   1:  PR[91,3] = PR[90,3] + 17.116;
   1:L PR[91] R[100]mm/sec CNT100;
   1:  PR[91,1] = PR[90,1] + -21.081;
   1:  PR[91,2] = PR[90,2] + -16.561;
   1:  PR[91,3] = PR[90,3] + 17.122;
   1:L PR[91] R[100]mm/sec CNT100;
   1:  PR[91,1] = PR[90,1] + -20.254;
   1:  PR[91,2] = PR[90,2] + -16.668;
   1:  PR[91,3] = PR[90,3] + 17.126;
   1:L PR[91] R[100]mm/sec CNT100;
   1:  PR[91,1] = PR[90,1] + -19.426;
   1:  PR[91,2] = PR[90,2] + -16.738;
   1:  PR[91,3] = PR[90,3] + 17.131;
   1:L PR[91] R[100]mm/sec CNT100;
   1:  PR[91,1] = PR[90,1] + -18.782;
   1:  PR[91,2] = PR[90,2] + -16.766;
   1:  PR[91,3] = PR[90,3] + 17.137;
   1:L PR[91] R[100]mm/sec CNT100;
   1:  PR[91,1] = PR[90,1] + -17.777;
   1:  PR[91,3] = PR[90,3] + 17.141;
   1:L PR[91] R[100]mm/sec CNT100;
   1:  PR[91,1] = PR[90,1] + -16.913;
   1:  PR[91,2] = PR[90,2] + -16.723;
   1:  PR[91,3] = PR[90,3] + 17.148;
   1:L PR[91] R[100]mm/sec CNT100;
   1:  PR[91,1] = PR[90,1] + -16.017;
   1:  PR[91,2] = PR[90,2] + -16.636;
   1:  PR[91,3] = PR[90,3] + 17.154;
   1:L PR[91] R[100]mm/sec CNT100;
   1:  PR[91,1] = PR[90,1] + -15.426;
   1:  PR[91,2] = PR[90,2] + -16.551;
   1:  PR[91,3] = PR[90,3] + 17.160;
   1:L PR[91] R[100]mm/sec CNT100;
   1:  PR[91,1] = PR[90,1] + -15.127;
   1:  PR[91,2] = PR[90,2] + -16.506;
   1:  PR[91,3] = PR[90,3] + 17.164;
   1:L PR[91] R[100]mm/sec CNT100;
   1:  PR[91,1] = PR[90,1] + -14.239;
   1:  PR[91,2] = PR[90,2] + -16.332;
   1:  PR[91,3] = PR[90,3] + 17.166;
   1:L PR[91] R[100]mm/sec CNT100;
   1:  PR[91,1] = PR[90,1] + -13.361;
   1:  PR[91,2] = PR[90,2] + -16.116;
   1:  PR[91,3] = PR[90,3] + 17.172;
   1:L PR[91] R[100]mm/sec CNT100;
   1:  PR[91,1] = PR[90,1] + -12.492;
   1:  PR[91,2] = PR[90,2] + -15.856;
   1:  PR[91,3] = PR[90,3] + 17.178;
   1:L PR[91] R[100]mm/sec CNT100;
   1:  PR[91,1] = PR[90,1] + -11.634;
   1:  PR[91,2] = PR[90,2] + -15.552;
   1:  PR[91,3] = PR[90,3] + 17.184;
   1:L PR[91] R[100]mm/sec CNT100;
   1:  PR[91,1] = PR[90,1] + -10.935;
   1:  PR[91,2] = PR[90,2] + -15.269;
   1:  PR[91,3] = PR[90,3] + 17.190;
   1:L PR[91] R[100]mm/sec CNT100;
   1:  PR[91,1] = PR[90,1] + -9.954;
   1:  PR[91,2] = PR[90,2] + -14.819;
   1:  PR[91,3] = PR[90,3] + 17.196;
   1:L PR[91] R[100]mm/sec CNT100;
   1:  PR[91,1] = PR[90,1] + -9.144;
   1:  PR[91,2] = PR[90,2] + -14.392;
   1:  PR[91,3] = PR[90,3] + 17.203;
   1:L PR[91] R[100]mm/sec CNT100;
   1:  PR[91,1] = PR[90,1] + -8.357;
   1:  PR[91,2] = PR[90,2] + -13.925;
   1:  PR[91,3] = PR[90,3] + 17.209;
   1:L PR[91] R[100]mm/sec CNT100;
   1:  PR[91,1] = PR[90,1] + -7.509;
   1:  PR[91,2] = PR[90,2] + -13.359;
   1:  PR[91,3] = PR[90,3] + 17.215;
   1:L PR[91] R[100]mm/sec CNT100;
   1:  PR[91,1] = PR[90,1] + -6.849;
   1:  PR[91,2] = PR[90,2] + -12.872;
   1:  PR[91,3] = PR[90,3] + 17.222;
   1:L PR[91] R[100]mm/sec CNT100;
   1:  PR[91,1] = PR[90,1] + -6.250;
   1:  PR[91,2] = PR[90,2] + -12.386;
   1:  PR[91,3] = PR[90,3] + 17.228;
   1:L PR[91] R[100]mm/sec CNT100;
   1:  PR[91,1] = PR[90,1] + -5.436;
   1:  PR[91,2] = PR[90,2] + -11.654;
   1:  PR[91,3] = PR[90,3] + 17.233;
   1:L PR[91] R[100]mm/sec CNT100;
   1:  PR[91,1] = PR[90,1] + -4.791;
   1:  PR[91,2] = PR[90,2] + -11.003;
   1:  PR[91,3] = PR[90,3] + 17.240;
   1:L PR[91] R[100]mm/sec CNT100;
   1:  PR[91,1] = PR[90,1] + -4.009;
   1:  PR[91,2] = PR[90,2] + -10.107;
   1:  PR[91,3] = PR[90,3] + 17.246;
   1:L PR[91] R[100]mm/sec CNT100;
   1:  PR[91,1] = PR[90,1] + -3.615;
   1:  PR[91,2] = PR[90,2] + -9.607;
   1:  PR[91,3] = PR[90,3] + 17.254;
   1:L PR[91] R[100]mm/sec CNT100;
   1:  PR[91,1] = PR[90,1] + -3.087;
   1:  PR[91,2] = PR[90,2] + -8.866;
   1:  PR[91,3] = PR[90,3] + 17.259;
   1:L PR[91] R[100]mm/sec CNT100;
   1:  PR[91,1] = PR[90,1] + -2.404;
   1:  PR[91,2] = PR[90,2] + -7.817;
   1:  PR[91,3] = PR[90,3] + 17.265;
   1:L PR[91] R[100]mm/sec CNT100;
   1:  PR[91,1] = PR[90,1] + -2.128;
   1:  PR[91,2] = PR[90,2] + -7.504;
   1:  PR[91,3] = PR[90,3] + 17.273;
   1:L PR[91] R[100]mm/sec CNT100;
   1:  PR[91,1] = PR[90,1] + -1.868;
   1:  PR[91,2] = PR[90,2] + -7.270;
   1:  PR[91,3] = PR[90,3] + 17.276;
   1:L PR[91] R[100]mm/sec CNT100;
   1:  PR[91,1] = PR[90,1] + -1.488;
   1:  PR[91,2] = PR[90,2] + -7.006;
   1:  PR[91,3] = PR[90,3] + 17.279;
   1:L PR[91] R[100]mm/sec CNT100;
   1:  PR[91,1] = PR[90,1] + -1.122;
   1:  PR[91,2] = PR[90,2] + -6.827;
   1:  PR[91,3] = PR[90,3] + 17.282;
   1:L PR[91] R[100]mm/sec CNT100;
   1:  PR[91,1] = PR[90,1] + -0.732;
   1:  PR[91,2] = PR[90,2] + -6.702;
   1:  PR[91,3] = PR[90,3] + 17.284;
   1:L PR[91] R[100]mm/sec CNT100;
   1:  PR[91,1] = PR[90,1] + -0.326;
   1:  PR[91,2] = PR[90,2] + -6.637;
   1:  PR[91,3] = PR[90,3] + 17.287;
   1:L PR[91] R[100]mm/sec CNT100;
   1:  PR[91] = PR[90];
   1:  PR[91,1] = PR[90,1] + 0.284;
   1:  PR[91,2] = PR[90,2] + -7.601;
   1:  PR[91,3] = PR[90,3] + 18.620;
   1:L PR[91] R[100]mm/sec CNT100;
   1:  PR[91,1] = PR[90,1] + 0.694;
   1:  PR[91,2] = PR[90,2] + -7.696;
   1:  PR[91,3] = PR[90,3] + 17.293;
   1:L PR[91] R[100]mm/sec CNT100;
   1:  PR[91,1] = PR[90,1] + 1.100;
   1:  PR[91,2] = PR[90,2] + -7.860;
   1:  PR[91,3] = PR[90,3] + 17.296;
   1:L PR[91] R[100]mm/sec CNT100;
   1:  PR[91,1] = PR[90,1] + 1.486;
   1:  PR[91,2] = PR[90,2] + -8.091;
   1:  PR[91,3] = PR[90,3] + 17.299;
   1:L PR[91] R[100]mm/sec CNT100;
   1:  PR[91,1] = PR[90,1] + 1.818;
   1:  PR[91,2] = PR[90,2] + -8.361;
   1:  PR[91,3] = PR[90,3] + 17.302;
   1:L PR[91] R[100]mm/sec CNT100;
   1:  PR[91,1] = PR[90,1] + 2.106;
   1:  PR[91,2] = PR[90,2] + -8.665;
   1:  PR[91,3] = PR[90,3] + 17.305;
   1:L PR[91] R[100]mm/sec CNT100;
   1:  PR[91,1] = PR[90,1] + 2.719;
   1:  PR[91,2] = PR[90,2] + -9.517;
   1:  PR[91,3] = PR[90,3] + 17.308;
   1:L PR[91] R[100]mm/sec CNT100;
   1:  PR[91,1] = PR[90,1] + 3.195;
   1:  PR[91,2] = PR[90,2] + -10.128;
   1:  PR[91,3] = PR[90,3] + 17.315;
   1:L PR[91] R[100]mm/sec CNT100;
   1:  PR[91,1] = PR[90,1] + 3.745;
   1:  PR[91,2] = PR[90,2] + -10.769;
   1:  PR[91,3] = PR[90,3] + 17.320;
   1:L PR[91] R[100]mm/sec CNT100;
   1:  PR[91,1] = PR[90,1] + 4.374;
   1:  PR[91,2] = PR[90,2] + -11.433;
   1:  PR[91,3] = PR[90,3] + 17.326;
   1:L PR[91] R[100]mm/sec CNT100;
   1:  PR[91,1] = PR[90,1] + 5.041;
   1:  PR[91,2] = PR[90,2] + -12.066;
   1:  PR[91,3] = PR[90,3] + 17.332;
   1:L PR[91] R[100]mm/sec CNT100;
   1:  PR[91,1] = PR[90,1] + 5.742;
   1:  PR[91,2] = PR[90,2] + -12.665;
   1:  PR[91,3] = PR[90,3] + 17.338;
   1:L PR[91] R[100]mm/sec CNT100;
   1:  PR[91,1] = PR[90,1] + 6.083;
   1:  PR[91,2] = PR[90,2] + -12.930;
   1:  PR[91,3] = PR[90,3] + 17.345;
   1:L PR[91] R[100]mm/sec CNT100;
   1:  PR[91,1] = PR[90,1] + 6.469;
   1:  PR[91,2] = PR[90,2] + -13.223;
   1:  PR[91,3] = PR[90,3] + 17.348;
   1:L PR[91] R[100]mm/sec CNT100;
   1:  PR[91,1] = PR[90,1] + 7.229;
   1:  PR[91,2] = PR[90,2] + -13.748;
   1:  PR[91,3] = PR[90,3] + 17.351;
   1:L PR[91] R[100]mm/sec CNT100;
   1:  PR[91,1] = PR[90,1] + 8.026;
   1:  PR[91,2] = PR[90,2] + -14.239;
   1:  PR[91,3] = PR[90,3] + 17.357;
   1:L PR[91] R[100]mm/sec CNT100;
   1:  PR[91,1] = PR[90,1] + 8.853;
   1:  PR[91,2] = PR[90,2] + -14.696;
   1:  PR[91,3] = PR[90,3] + 17.364;
   1:L PR[91] R[100]mm/sec CNT100;
   1:  PR[91,1] = PR[90,1] + 9.431;
   1:  PR[91,2] = PR[90,2] + -14.983;
   1:  PR[91,3] = PR[90,3] + 17.370;
   1:L PR[91] R[100]mm/sec CNT100;
   1:  PR[91,1] = PR[90,1] + 10.170;
   1:  PR[91,2] = PR[90,2] + -15.316;
   1:  PR[91,3] = PR[90,3] + 17.375;
   1:L PR[91] R[100]mm/sec CNT100;
   1:  PR[91,1] = PR[90,1] + 10.927;
   1:  PR[91,2] = PR[90,2] + -15.619;
   1:  PR[91,3] = PR[90,3] + 17.380;
   1:L PR[91] R[100]mm/sec CNT100;
   1:  PR[91,1] = PR[90,1] + 11.523;
   1:  PR[91,2] = PR[90,2] + -15.832;
   1:  PR[91,3] = PR[90,3] + 17.386;
   1:L PR[91] R[100]mm/sec CNT100;
   1:  PR[91,1] = PR[90,1] + 12.486;
   1:  PR[91,2] = PR[90,2] + -16.130;
   1:  PR[91,3] = PR[90,3] + 17.390;
   1:L PR[91] R[100]mm/sec CNT100;
   1:  PR[91,1] = PR[90,1] + 13.368;
   1:  PR[91,2] = PR[90,2] + -16.357;
   1:  PR[91,3] = PR[90,3] + 17.397;
   1:L PR[91] R[100]mm/sec CNT100;
   1:  PR[91,1] = PR[90,1] + 14.012;
   1:  PR[91,2] = PR[90,2] + -16.491;
   1:  PR[91,3] = PR[90,3] + 17.403;
   1:L PR[91] R[100]mm/sec CNT100;
   1:  PR[91,1] = PR[90,1] + 15.181;
   1:  PR[91,2] = PR[90,2] + -16.684;
   1:  PR[91,3] = PR[90,3] + 17.408;
   1:L PR[91] R[100]mm/sec CNT100;
   1:  PR[91,1] = PR[90,1] + 16.352;
   1:  PR[91,2] = PR[90,2] + -16.797;
   1:  PR[91,3] = PR[90,3] + 17.416;
   1:L PR[91] R[100]mm/sec CNT100;
   1:  PR[91,1] = PR[90,1] + 17.007;
   1:  PR[91,2] = PR[90,2] + -16.833;
   1:  PR[91,3] = PR[90,3] + 17.424;
   1:L PR[91] R[100]mm/sec CNT100;
   1:  PR[91,1] = PR[90,1] + 17.921;
   1:  PR[91,2] = PR[90,2] + -16.841;
   1:  PR[91,3] = PR[90,3] + 17.428;
   1:L PR[91] R[100]mm/sec CNT100;
   1:  PR[91,1] = PR[90,1] + 18.825;
   1:  PR[91,2] = PR[90,2] + -16.806;
   1:  PR[91,3] = PR[90,3] + 17.435;
   1:L PR[91] R[100]mm/sec CNT100;
   1:  PR[91,1] = PR[90,1] + 19.474;
   1:  PR[91,2] = PR[90,2] + -16.751;
   1:  PR[91,3] = PR[90,3] + 17.441;
   1:L PR[91] R[100]mm/sec CNT100;
   1:  PR[91,1] = PR[90,1] + 20.614;
   1:  PR[91,2] = PR[90,2] + -16.607;
   1:  PR[91,3] = PR[90,3] + 17.445;
   1:L PR[91] R[100]mm/sec CNT100;
   1:  PR[91,1] = PR[90,1] + 21.491;
   1:  PR[91,2] = PR[90,2] + -16.445;
   1:  PR[91,3] = PR[90,3] + 17.453;
   1:L PR[91] R[100]mm/sec CNT100;
   1:  PR[91,1] = PR[90,1] + 22.358;
   1:  PR[91,2] = PR[90,2] + -16.242;
   1:  PR[91,3] = PR[90,3] + 17.459;
   1:L PR[91] R[100]mm/sec CNT100;
   1:  PR[91,1] = PR[90,1] + 23.212;
   1:  PR[91,2] = PR[90,2] + -15.997;
   1:  PR[91,3] = PR[90,3] + 17.466;
   1:L PR[91] R[100]mm/sec CNT100;
   1:  PR[91,1] = PR[90,1] + 24.055;
   1:  PR[91,2] = PR[90,2] + -15.712;
   1:  PR[91,3] = PR[90,3] + 17.472;
   1:L PR[91] R[100]mm/sec CNT100;
   1:  PR[91,1] = PR[90,1] + 24.829;
   1:  PR[91,2] = PR[90,2] + -15.409;
   1:  PR[91,3] = PR[90,3] + 17.478;
   1:L PR[91] R[100]mm/sec CNT100;
   1:  PR[91,1] = PR[90,1] + 25.593;
   1:  PR[91,2] = PR[90,2] + -15.069;
   1:  PR[91,3] = PR[90,3] + 17.483;
   1:L PR[91] R[100]mm/sec CNT100;
   1:  PR[91,1] = PR[90,1] + 26.342;
   1:  PR[91,2] = PR[90,2] + -14.694;
   1:  PR[91,3] = PR[90,3] + 17.489;
   1:L PR[91] R[100]mm/sec CNT100;
   1:  PR[91,1] = PR[90,1] + 27.074;
   1:  PR[91,2] = PR[90,2] + -14.284;
   1:  PR[91,3] = PR[90,3] + 17.495;
   1:L PR[91] R[100]mm/sec CNT100;
   1:  PR[91,1] = PR[90,1] + 27.788;
   1:  PR[91,2] = PR[90,2] + -13.840;
   1:  PR[91,3] = PR[90,3] + 17.501;
   1:L PR[91] R[100]mm/sec CNT100;
   1:  PR[91,1] = PR[90,1] + 28.480;
   1:  PR[91,2] = PR[90,2] + -13.362;
   1:  PR[91,3] = PR[90,3] + 17.506;
   1:L PR[91] R[100]mm/sec CNT100;
   1:  PR[91,1] = PR[90,1] + 29.151;
   1:  PR[91,2] = PR[90,2] + -12.851;
   1:  PR[91,3] = PR[90,3] + 17.512;
   1:L PR[91] R[100]mm/sec CNT100;
   1:  PR[91,1] = PR[90,1] + 29.796;
   1:  PR[91,2] = PR[90,2] + -12.308;
   1:  PR[91,3] = PR[90,3] + 17.518;
   1:L PR[91] R[100]mm/sec CNT100;
   1:  PR[91,1] = PR[90,1] + 30.416;
   1:  PR[91,2] = PR[90,2] + -11.732;
   1:  PR[91,3] = PR[90,3] + 17.524;
   1:L PR[91] R[100]mm/sec CNT100;
   1:  PR[91,1] = PR[90,1] + 31.008;
   1:  PR[91,2] = PR[90,2] + -11.127;
   1:  PR[91,3] = PR[90,3] + 17.530;
   1:L PR[91] R[100]mm/sec CNT100;
   1:  PR[91,1] = PR[90,1] + 31.571;
   1:  PR[91,2] = PR[90,2] + -10.489;
   1:  PR[91,3] = PR[90,3] + 17.535;
   1:L PR[91] R[100]mm/sec CNT100;
   1:  PR[91,1] = PR[90,1] + 32.107;
   1:  PR[91,2] = PR[90,2] + -9.815;
   1:  PR[91,3] = PR[90,3] + 17.541;
   1:L PR[91] R[100]mm/sec CNT100;
   1:  PR[91,1] = PR[90,1] + 32.609;
   1:  PR[91,2] = PR[90,2] + -9.116;
   1:  PR[91,3] = PR[90,3] + 17.547;
   1:L PR[91] R[100]mm/sec CNT100;
   1:  PR[91,1] = PR[90,1] + 33.075;
   1:  PR[91,2] = PR[90,2] + -8.395;
   1:  PR[91,3] = PR[90,3] + 17.553;
   1:L PR[91] R[100]mm/sec CNT100;
   1:  PR[91,1] = PR[90,1] + 33.503;
   1:  PR[91,2] = PR[90,2] + -7.655;
   1:  PR[91,3] = PR[90,3] + 17.559;
   1:L PR[91] R[100]mm/sec CNT100;
   1:  PR[91,1] = PR[90,1] + 33.894;
   1:  PR[91,2] = PR[90,2] + -6.899;
   1:  PR[91,3] = PR[90,3] + 17.565;
   1:L PR[91] R[100]mm/sec CNT100;
   1:  PR[91,1] = PR[90,1] + 34.245;
   1:  PR[91,2] = PR[90,2] + -6.131;
   1:  PR[91,3] = PR[90,3] + 17.571;
   1:L PR[91] R[100]mm/sec CNT100;
   1:  PR[91,1] = PR[90,1] + 34.557;
   1:  PR[91,2] = PR[90,2] + -5.354;
   1:  PR[91,3] = PR[90,3] + 17.576;
   1:L PR[91] R[100]mm/sec CNT100;
   1:  PR[91,1] = PR[90,1] + 34.828;
   1:  PR[91,2] = PR[90,2] + -4.568;
   1:  PR[91,3] = PR[90,3] + 17.582;
   1:L PR[91] R[100]mm/sec CNT100;
   1:  PR[91,1] = PR[90,1] + 35.058;
   1:  PR[91,2] = PR[90,2] + -3.774;
   1:  PR[91,3] = PR[90,3] + 17.588;
   1:L PR[91] R[100]mm/sec CNT100;
   1:  PR[91,1] = PR[90,1] + 35.246;
   1:  PR[91,2] = PR[90,2] + -2.968;
   1:  PR[91,3] = PR[90,3] + 17.593;
   1:L PR[91] R[100]mm/sec CNT100;
   1:  PR[91,1] = PR[90,1] + 35.394;
   1:  PR[91,2] = PR[90,2] + -2.148;
   1:  PR[91,3] = PR[90,3] + 17.599;
   1:L PR[91] R[100]mm/sec CNT100;
   1:  PR[91,1] = PR[90,1] + 35.499;
   1:  PR[91,2] = PR[90,2] + -1.310;
   1:  PR[91,3] = PR[90,3] + 17.605;
   1:L PR[91] R[100]mm/sec CNT100;
   1:  PR[91,1] = PR[90,1] + 35.563;
   1:  PR[91,2] = PR[90,2] + -0.453;
   1:  PR[91,3] = PR[90,3] + 17.611;
   1:L PR[91] R[100]mm/sec CNT100;
   1:  PR[91,1] = PR[90,1] + 35.585;
   1:  PR[91,2] = PR[90,2] + 0.428;
   1:  PR[91,3] = PR[90,3] + 17.616;
   1:L PR[91] R[100]mm/sec CNT100;
   1:  PR[91,1] = PR[90,1] + 35.563;
   1:  PR[91,2] = PR[90,2] + 1.308;
   1:  PR[91,3] = PR[90,3] + 17.623;
   1:L PR[91] R[100]mm/sec CNT100;
   1:  PR[91,1] = PR[90,1] + 35.499;
   1:  PR[91,2] = PR[90,2] + 2.165;
   1:  PR[91,3] = PR[90,3] + 17.629;
   1:L PR[91] R[100]mm/sec CNT100;
   1:  PR[91,1] = PR[90,1] + 35.394;
   1:  PR[91,2] = PR[90,2] + 3.003;
   1:  PR[91,3] = PR[90,3] + 17.634;
   1:L PR[91] R[100]mm/sec CNT100;
   1:  PR[91,1] = PR[90,1] + 35.246;
   1:  PR[91,2] = PR[90,2] + 3.823;
   1:  PR[91,3] = PR[90,3] + 17.640;
   1:L PR[91] R[100]mm/sec CNT100;
   1:  PR[91,1] = PR[90,1] + 35.058;
   1:  PR[91,2] = PR[90,2] + 4.629;
   1:  PR[91,3] = PR[90,3] + 17.646;
   1:L PR[91] R[100]mm/sec CNT100;
   1:  PR[91,1] = PR[90,1] + 34.828;
   1:  PR[91,2] = PR[90,2] + 5.424;
   1:  PR[91,3] = PR[90,3] + 17.652;
   1:L PR[91] R[100]mm/sec CNT100;
   1:  PR[91,1] = PR[90,1] + 34.557;
   1:  PR[91,2] = PR[90,2] + 6.209;
   1:  PR[91,3] = PR[90,3] + 17.657;
   1:L PR[91] R[100]mm/sec CNT100;
   1:  PR[91,1] = PR[90,1] + 34.245;
   1:  PR[91,2] = PR[90,2] + 6.986;
   1:  PR[91,3] = PR[90,3] + 17.663;
   1:L PR[91] R[100]mm/sec CNT100;
   1:  PR[91,1] = PR[90,1] + 33.894;
   1:  PR[91,2] = PR[90,2] + 7.754;
   1:  PR[91,3] = PR[90,3] + 17.669;
   1:L PR[91] R[100]mm/sec CNT100;
   1:  PR[91,1] = PR[90,1] + 33.503;
   1:  PR[91,2] = PR[90,2] + 8.510;
   1:  PR[91,3] = PR[90,3] + 17.675;
   1:L PR[91] R[100]mm/sec CNT100;
   1:  PR[91,1] = PR[90,1] + 33.074;
   1:  PR[91,2] = PR[90,2] + 9.250;
   1:  PR[91,3] = PR[90,3] + 17.680;
   1:L PR[91] R[100]mm/sec CNT100;
   1:  PR[91,1] = PR[90,1] + 32.609;
   1:  PR[91,2] = PR[90,2] + 9.972;
   1:  PR[91,3] = PR[90,3] + 17.686;
   1:L PR[91] R[100]mm/sec CNT100;
   1:  PR[91,1] = PR[90,1] + 32.107;
   1:  PR[91,2] = PR[90,2] + 10.670;
   1:  PR[91,3] = PR[90,3] + 17.692;
   1:L PR[91] R[100]mm/sec CNT100;
   1:  PR[91,1] = PR[90,1] + 31.565;
   1:  PR[91,2] = PR[90,2] + 11.351;
   1:  PR[91,3] = PR[90,3] + 17.698;
   1:L PR[91] R[100]mm/sec CNT100;
   1:  PR[91,1] = PR[90,1] + 31.009;
   1:  PR[91,2] = PR[90,2] + 11.980;
   1:  PR[91,3] = PR[90,3] + 17.704;
   1:L PR[91] R[100]mm/sec CNT100;
   1:  PR[91,1] = PR[90,1] + 30.326;
   1:  PR[91,2] = PR[90,2] + 12.673;
   1:  PR[91,3] = PR[90,3] + 17.710;
   1:L PR[91] R[100]mm/sec CNT100;
   1:  PR[91,1] = PR[90,1] + 29.797;
   1:  PR[91,2] = PR[90,2] + 13.162;
   1:  PR[91,3] = PR[90,3] + 17.716;
   1:L PR[91] R[100]mm/sec CNT100;
   1:  PR[91,1] = PR[90,1] + 29.151;
   1:  PR[91,2] = PR[90,2] + 13.706;
   1:  PR[91,3] = PR[90,3] + 17.721;
   1:L PR[91] R[100]mm/sec CNT100;
   1:  PR[91,1] = PR[90,1] + 28.479;
   1:  PR[91,2] = PR[90,2] + 14.218;
   1:  PR[91,3] = PR[90,3] + 17.727;
   1:L PR[91] R[100]mm/sec CNT100;
   1:  PR[91,1] = PR[90,1] + 28.191;
   1:  PR[91,2] = PR[90,2] + 14.420;
   1:  PR[91,3] = PR[90,3] + 17.733;
   1:L PR[91] R[100]mm/sec CNT100;
   1:  PR[91,1] = PR[90,1] + 27.789;
   1:  PR[91,2] = PR[90,2] + 14.694;
   1:  PR[91,3] = PR[90,3] + 17.735;
   1:L PR[91] R[100]mm/sec CNT100;
   1:  PR[91,1] = PR[90,1] + 27.074;
   1:  PR[91,2] = PR[90,2] + 15.139;
   1:  PR[91,3] = PR[90,3] + 17.739;
   1:L PR[91] R[100]mm/sec CNT100;
   1:  PR[91,1] = PR[90,1] + 26.341;
   1:  PR[91,2] = PR[90,2] + 15.550;
   1:  PR[91,3] = PR[90,3] + 17.744;
   1:L PR[91] R[100]mm/sec CNT100;
   1:  PR[91,1] = PR[90,1] + 25.781;
   1:  PR[91,2] = PR[90,2] + 15.832;
   1:  PR[91,3] = PR[90,3] + 17.750;
   1:L PR[91] R[100]mm/sec CNT100;
   1:  PR[91,1] = PR[90,1] + 24.827;
   1:  PR[91,2] = PR[90,2] + 16.265;
   1:  PR[91,3] = PR[90,3] + 17.754;
   1:L PR[91] R[100]mm/sec CNT100;
   1:  PR[91,1] = PR[90,1] + 24.051;
   1:  PR[91,2] = PR[90,2] + 16.569;
   1:  PR[91,3] = PR[90,3] + 17.762;
   1:L PR[91] R[100]mm/sec CNT100;
   1:  PR[91,1] = PR[90,1] + 23.212;
   1:  PR[91,2] = PR[90,2] + 16.853;
   1:  PR[91,3] = PR[90,3] + 17.767;
   1:L PR[91] R[100]mm/sec CNT100;
   1:  PR[91,1] = PR[90,1] + 22.358;
   1:  PR[91,2] = PR[90,2] + 17.097;
   1:  PR[91,3] = PR[90,3] + 17.773;
   1:L PR[91] R[100]mm/sec CNT100;
   1:  PR[91,1] = PR[90,1] + 21.490;
   1:  PR[91,2] = PR[90,2] + 17.301;
   1:  PR[91,3] = PR[90,3] + 17.780;
   1:L PR[91] R[100]mm/sec CNT100;
   1:  PR[91,1] = PR[90,1] + 21.028;
   1:  PR[91,2] = PR[90,2] + 17.388;
   1:  PR[91,3] = PR[90,3] + 17.786;
   1:L PR[91] R[100]mm/sec CNT100;
   1:  PR[91,1] = PR[90,1] + 20.612;
   1:  PR[91,2] = PR[90,2] + 17.463;
   1:  PR[91,3] = PR[90,3] + 17.789;
   1:L PR[91] R[100]mm/sec CNT100;
   1:  PR[91,1] = PR[90,1] + 19.722;
   1:  PR[91,2] = PR[90,2] + 17.583;
   1:  PR[91,3] = PR[90,3] + 17.792;
   1:L PR[91] R[100]mm/sec CNT100;
   1:  PR[91,1] = PR[90,1] + 18.825;
   1:  PR[91,2] = PR[90,2] + 17.661;
   1:  PR[91,3] = PR[90,3] + 17.798;
   1:L PR[91] R[100]mm/sec CNT100;
   1:  PR[91,1] = PR[90,1] + 17.918;
   1:  PR[91,2] = PR[90,2] + 17.696;
   1:  PR[91,3] = PR[90,3] + 17.804;
   1:L PR[91] R[100]mm/sec CNT100;
   1:  PR[91,1] = PR[90,1] + 17.008;
   1:  PR[91,2] = PR[90,2] + 17.688;
   1:  PR[91,3] = PR[90,3] + 17.810;
   1:L PR[91] R[100]mm/sec CNT100;
   1:  PR[91,1] = PR[90,1] + 16.094;
   1:  PR[91,2] = PR[90,2] + 17.636;
   1:  PR[91,3] = PR[90,3] + 17.817;
   1:L PR[91] R[100]mm/sec CNT100;
   1:  PR[91,1] = PR[90,1] + 15.184;
   1:  PR[91,2] = PR[90,2] + 17.539;
   1:  PR[91,3] = PR[90,3] + 17.823;
   1:L PR[91] R[100]mm/sec CNT100;
   1:  PR[91,1] = PR[90,1] + 14.012;
   1:  PR[91,2] = PR[90,2] + 17.346;
   1:  PR[91,3] = PR[90,3] + 17.829;
   1:L PR[91] R[100]mm/sec CNT100;
   1:  PR[91,1] = PR[90,1] + 13.368;
   1:  PR[91,2] = PR[90,2] + 17.212;
   1:  PR[91,3] = PR[90,3] + 17.837;
   1:L PR[91] R[100]mm/sec CNT100;
   1:  PR[91,1] = PR[90,1] + 12.462;
   1:  PR[91,2] = PR[90,2] + 16.979;
   1:  PR[91,3] = PR[90,3] + 17.842;
   1:L PR[91] R[100]mm/sec CNT100;
   1:  PR[91,1] = PR[90,1] + 11.698;
   1:  PR[91,2] = PR[90,2] + 16.745;
   1:  PR[91,3] = PR[90,3] + 17.848;
   1:L PR[91] R[100]mm/sec CNT100;
   1:  PR[91,1] = PR[90,1] + 10.925;
   1:  PR[91,2] = PR[90,2] + 16.473;
   1:  PR[91,3] = PR[90,3] + 17.854;
   1:L PR[91] R[100]mm/sec CNT100;
   1:  PR[91,1] = PR[90,1] + 10.168;
   1:  PR[91,2] = PR[90,2] + 16.170;
   1:  PR[91,3] = PR[90,3] + 17.859;
   1:L PR[91] R[100]mm/sec CNT100;
   1:  PR[91,1] = PR[90,1] + 9.721;
   1:  PR[91,2] = PR[90,2] + 15.974;
   1:  PR[91,3] = PR[90,3] + 17.865;
   1:L PR[91] R[100]mm/sec CNT100;
   1:  PR[91,1] = PR[90,1] + 8.712;
   1:  PR[91,2] = PR[90,2] + 15.477;
   1:  PR[91,3] = PR[90,3] + 17.868;
   1:L PR[91] R[100]mm/sec CNT100;
   1:  PR[91,1] = PR[90,1] + 8.015;
   1:  PR[91,2] = PR[90,2] + 15.088;
   1:  PR[91,3] = PR[90,3] + 17.876;
   1:L PR[91] R[100]mm/sec CNT100;
   1:  PR[91,1] = PR[90,1] + 7.356;
   1:  PR[91,2] = PR[90,2] + 14.683;
   1:  PR[91,3] = PR[90,3] + 17.881;
   1:L PR[91] R[100]mm/sec CNT100;
   1:  PR[91,1] = PR[90,1] + 6.469;
   1:  PR[91,2] = PR[90,2] + 14.078;
   1:  PR[91,3] = PR[90,3] + 17.887;
   1:L PR[91] R[100]mm/sec CNT100;
   1:  PR[91,1] = PR[90,1] + 5.738;
   1:  PR[91,2] = PR[90,2] + 13.517;
   1:  PR[91,3] = PR[90,3] + 17.894;
   1:L PR[91] R[100]mm/sec CNT100;
   1:  PR[91,1] = PR[90,1] + 5.477;
   1:  PR[91,2] = PR[90,2] + 13.298;
   1:  PR[91,3] = PR[90,3] + 17.900;
   1:L PR[91] R[100]mm/sec CNT100;
   1:  PR[91,1] = PR[90,1] + 5.042;
   1:  PR[91,2] = PR[90,2] + 12.922;
   1:  PR[91,3] = PR[90,3] + 17.903;
   1:L PR[91] R[100]mm/sec CNT100;
   1:  PR[91,1] = PR[90,1] + 4.374;
   1:  PR[91,2] = PR[90,2] + 12.287;
   1:  PR[91,3] = PR[90,3] + 17.907;
   1:L PR[91] R[100]mm/sec CNT100;
   1:  PR[91,1] = PR[90,1] + 3.745;
   1:  PR[91,2] = PR[90,2] + 11.624;
   1:  PR[91,3] = PR[90,3] + 17.913;
   1:L PR[91] R[100]mm/sec CNT100;
   1:  PR[91,1] = PR[90,1] + 3.195;
   1:  PR[91,2] = PR[90,2] + 10.983;
   1:  PR[91,3] = PR[90,3] + 17.919;
   1:L PR[91] R[100]mm/sec CNT100;
   1:  PR[91,1] = PR[90,1] + 2.719;
   1:  PR[91,2] = PR[90,2] + 10.372;
   1:  PR[91,3] = PR[90,3] + 17.925;
   1:L PR[91] R[100]mm/sec CNT100;
   1:  PR[91,1] = PR[90,1] + 2.105;
   1:  PR[91,2] = PR[90,2] + 9.520;
   1:  PR[91,3] = PR[90,3] + 17.930;
   1:L PR[91] R[100]mm/sec CNT100;
   1:  PR[91,1] = PR[90,1] + 1.817;
   1:  PR[91,2] = PR[90,2] + 9.215;
   1:  PR[91,3] = PR[90,3] + 17.937;
   1:L PR[91] R[100]mm/sec CNT100;
   1:  PR[91,1] = PR[90,1] + 1.485;
   1:  PR[91,2] = PR[90,2] + 8.946;
   1:  PR[91,3] = PR[90,3] + 17.940;
   1:L PR[91] R[100]mm/sec CNT100;
   1:  PR[91,1] = PR[90,1] + 1.096;
   1:  PR[91,2] = PR[90,2] + 8.713;
   1:  PR[91,3] = PR[90,3] + 17.943;
   1:L PR[91] R[100]mm/sec CNT100;
   1:  PR[91,1] = PR[90,1] + 0.664;
   1:  PR[91,2] = PR[90,2] + 8.544;
   1:  PR[91,3] = PR[90,3] + 17.946;
   1:L PR[91] R[100]mm/sec CNT100;
   1:  PR[91,1] = PR[90,1] + 0.312;
   1:  PR[91,2] = PR[90,2] + 8.461;
   1:  PR[91,3] = PR[90,3] + 17.950;
   1:L PR[91] R[100]mm/sec CNT100;
   1:  PR[91,1] = PR[90,1] + -0.116;
   1:  PR[91,2] = PR[90,2] + 8.426;
   1:  PR[91,3] = PR[90,3] + 17.952;
   1:L PR[91] R[100]mm/sec CNT100;
   1:  PR[91,1] = PR[90,1] + -0.520;
   1:  PR[91,2] = PR[90,2] + 8.457;
   1:  PR[91,3] = PR[90,3] + 17.955;
   1:L PR[91] R[100]mm/sec CNT100;
   1:  PR[91,1] = PR[90,1] + -0.929;
   1:  PR[91,2] = PR[90,2] + 8.552;
   1:  PR[91,3] = PR[90,3] + 17.958;
   1:L PR[91] R[100]mm/sec CNT100;
   1:  PR[91,1] = PR[90,1] + -1.333;
   1:  PR[91,2] = PR[90,2] + 8.716;
   1:  PR[91,3] = PR[90,3] + 17.961;
   1:L PR[91] R[100]mm/sec CNT100;
   1:  PR[91,1] = PR[90,1] + -1.719;
   1:  PR[91,2] = PR[90,2] + 8.947;
   1:  PR[91,3] = PR[90,3] + 17.964;
   1:L PR[91] R[100]mm/sec CNT100;
   1:  PR[91,1] = PR[90,1] + -2.051;
   1:  PR[91,2] = PR[90,2] + 9.217;
   1:  PR[91,3] = PR[90,3] + 17.967;
   1:L PR[91] R[100]mm/sec CNT100;
   1:  PR[91,1] = PR[90,1] + -2.338;
   1:  PR[91,2] = PR[90,2] + 9.522;
   1:  PR[91,3] = PR[90,3] + 17.970;
   1:L PR[91] R[100]mm/sec CNT100;
   1:  PR[91,1] = PR[90,1] + -2.949;
   1:  PR[91,2] = PR[90,2] + 10.372;
   1:  PR[91,3] = PR[90,3] + 17.973;
   1:L PR[91] R[100]mm/sec CNT100;
   1:  PR[91,1] = PR[90,1] + -3.424;
   1:  PR[91,2] = PR[90,2] + 10.981;
   1:  PR[91,3] = PR[90,3] + 17.980;
   1:L PR[91] R[100]mm/sec CNT100;
   1:  PR[91,1] = PR[90,1] + -3.975;
   1:  PR[91,2] = PR[90,2] + 11.620;
   1:  PR[91,3] = PR[90,3] + 17.985;
   1:L PR[91] R[100]mm/sec CNT100;
   1:  PR[91,1] = PR[90,1] + -4.606;
   1:  PR[91,2] = PR[90,2] + 12.283;
   1:  PR[91,3] = PR[90,3] + 17.991;
   1:L PR[91] R[100]mm/sec CNT100;
   1:  PR[91,1] = PR[90,1] + -5.273;
   1:  PR[91,2] = PR[90,2] + 12.914;
   1:  PR[91,3] = PR[90,3] + 17.997;
   1:L PR[91] R[100]mm/sec CNT100;
   1:  PR[91,1] = PR[90,1] + -5.975;
   1:  PR[91,2] = PR[90,2] + 13.513;
   1:  PR[91,3] = PR[90,3] + 18.003;
   1:L PR[91] R[100]mm/sec CNT100;
   1:  PR[91,1] = PR[90,1] + -6.316;
   1:  PR[91,2] = PR[90,2] + 13.778;
   1:  PR[91,3] = PR[90,3] + 18.010;
   1:L PR[91] R[100]mm/sec CNT100;
   1:  PR[91,1] = PR[90,1] + -6.703;
   1:  PR[91,2] = PR[90,2] + 14.071;
   1:  PR[91,3] = PR[90,3] + 18.013;
   1:L PR[91] R[100]mm/sec CNT100;
   1:  PR[91,1] = PR[90,1] + -7.463;
   1:  PR[91,2] = PR[90,2] + 14.597;
   1:  PR[91,3] = PR[90,3] + 18.016;
   1:L PR[91] R[100]mm/sec CNT100;
   1:  PR[91,1] = PR[90,1] + -8.265;
   1:  PR[91,2] = PR[90,2] + 15.092;
   1:  PR[91,3] = PR[90,3] + 18.022;
   1:L PR[91] R[100]mm/sec CNT100;
   1:  PR[91,1] = PR[90,1] + -9.089;
   1:  PR[91,2] = PR[90,2] + 15.548;
   1:  PR[91,3] = PR[90,3] + 18.029;
   1:L PR[91] R[100]mm/sec CNT100;
   1:  PR[91,1] = PR[90,1] + -9.668;
   1:  PR[91,2] = PR[90,2] + 15.837;
   1:  PR[91,3] = PR[90,3] + 18.035;
   1:L PR[91] R[100]mm/sec CNT100;
   1:  PR[91,1] = PR[90,1] + -10.408;
   1:  PR[91,2] = PR[90,2] + 16.171;
   1:  PR[91,3] = PR[90,3] + 18.040;
   1:L PR[91] R[100]mm/sec CNT100;
   1:  PR[91,1] = PR[90,1] + -11.165;
   1:  PR[91,2] = PR[90,2] + 16.475;
   1:  PR[91,3] = PR[90,3] + 18.045;
   1:L PR[91] R[100]mm/sec CNT100;
   1:  PR[91,1] = PR[90,1] + -11.760;
   1:  PR[91,2] = PR[90,2] + 16.689;
   1:  PR[91,3] = PR[90,3] + 18.051;
   1:L PR[91] R[100]mm/sec CNT100;
   1:  PR[91,1] = PR[90,1] + -12.724;
   1:  PR[91,2] = PR[90,2] + 16.987;
   1:  PR[91,3] = PR[90,3] + 18.055;
   1:L PR[91] R[100]mm/sec CNT100;
   1:  PR[91,1] = PR[90,1] + -13.606;
   1:  PR[91,2] = PR[90,2] + 17.213;
   1:  PR[91,3] = PR[90,3] + 18.062;
   1:L PR[91] R[100]mm/sec CNT100;
   1:  PR[91,1] = PR[90,1] + -14.250;
   1:  PR[91,2] = PR[90,2] + 17.347;
   1:  PR[91,3] = PR[90,3] + 18.068;
   1:L PR[91] R[100]mm/sec CNT100;
   1:  PR[91,1] = PR[90,1] + -15.421;
   1:  PR[91,2] = PR[90,2] + 17.539;
   1:  PR[91,3] = PR[90,3] + 18.073;
   1:L PR[91] R[100]mm/sec CNT100;
   1:  PR[91,1] = PR[90,1] + -16.592;
   1:  PR[91,2] = PR[90,2] + 17.652;
   1:  PR[91,3] = PR[90,3] + 18.081;
   1:L PR[91] R[100]mm/sec CNT100;
   1:  PR[91,1] = PR[90,1] + -17.248;
   1:  PR[91,2] = PR[90,2] + 17.687;
   1:  PR[91,3] = PR[90,3] + 18.089;
   1:L PR[91] R[100]mm/sec CNT100;
   1:  PR[91,1] = PR[90,1] + -18.163;
   1:  PR[91,2] = PR[90,2] + 17.695;
   1:  PR[91,3] = PR[90,3] + 18.094;
   1:L PR[91] R[100]mm/sec CNT100;
   1:  PR[91,1] = PR[90,1] + -19.067;
   1:  PR[91,2] = PR[90,2] + 17.661;
   1:  PR[91,3] = PR[90,3] + 18.100;
   1:L PR[91] R[100]mm/sec CNT100;
   1:  PR[91,1] = PR[90,1] + -19.715;
   1:  PR[91,2] = PR[90,2] + 17.606;
   1:  PR[91,3] = PR[90,3] + 18.106;
   1:L PR[91] R[100]mm/sec CNT100;
   1:  PR[91,1] = PR[90,1] + -20.856;
   1:  PR[91,2] = PR[90,2] + 17.462;
   1:  PR[91,3] = PR[90,3] + 18.110;
   1:L PR[91] R[100]mm/sec CNT100;
   1:  PR[91,1] = PR[90,1] + -21.731;
   1:  PR[91,2] = PR[90,2] + 17.300;
   1:  PR[91,3] = PR[90,3] + 18.118;
   1:L PR[91] R[100]mm/sec CNT100;
   1:  PR[91,1] = PR[90,1] + -22.803;
   1:  PR[91,2] = PR[90,2] + 17.040;
   1:  PR[91,3] = PR[90,3] + 18.124;
   1:L PR[91] R[100]mm/sec CNT100;
   1:  PR[91,1] = PR[90,1] + -23.454;
   1:  PR[91,2] = PR[90,2] + 16.853;
   1:  PR[91,3] = PR[90,3] + 18.132;
   1:L PR[91] R[100]mm/sec CNT100;
   1:  PR[91,1] = PR[90,1] + -24.297;
   1:  PR[91,2] = PR[90,2] + 16.568;
   1:  PR[91,3] = PR[90,3] + 18.137;
   1:L PR[91] R[100]mm/sec CNT100;
   1:  PR[91,1] = PR[90,1] + -25.071;
   1:  PR[91,2] = PR[90,2] + 16.264;
   1:  PR[91,3] = PR[90,3] + 18.143;
   1:L PR[91] R[100]mm/sec CNT100;
   1:  PR[91,1] = PR[90,1] + -25.834;
   1:  PR[91,2] = PR[90,2] + 15.923;
   1:  PR[91,3] = PR[90,3] + 18.148;
   1:L PR[91] R[100]mm/sec CNT100;
   1:  PR[91,1] = PR[90,1] + -26.583;
   1:  PR[91,2] = PR[90,2] + 15.547;
   1:  PR[91,3] = PR[90,3] + 18.154;
   1:L PR[91] R[100]mm/sec CNT100;
   1:  PR[91,1] = PR[90,1] + -27.315;
   1:  PR[91,2] = PR[90,2] + 15.136;
   1:  PR[91,3] = PR[90,3] + 18.160;
   1:L PR[91] R[100]mm/sec CNT100;
   1:  PR[91,1] = PR[90,1] + -28.030;
   1:  PR[91,2] = PR[90,2] + 14.690;
   1:  PR[91,3] = PR[90,3] + 18.166;
   1:L PR[91] R[100]mm/sec CNT100;
   1:  PR[91,1] = PR[90,1] + -28.432;
   1:  PR[91,2] = PR[90,2] + 14.416;
   1:  PR[91,3] = PR[90,3] + 18.171;
   1:L PR[91] R[100]mm/sec CNT100;
   1:  PR[91,1] = PR[90,1] + -28.720;
   1:  PR[91,2] = PR[90,2] + 14.214;
   1:  PR[91,3] = PR[90,3] + 18.175;
   1:L PR[91] R[100]mm/sec CNT100;
   1:  PR[91,1] = PR[90,1] + -29.392;
   1:  PR[91,2] = PR[90,2] + 13.702;
   1:  PR[91,3] = PR[90,3] + 18.177;
   1:L PR[91] R[100]mm/sec CNT100;
   1:  PR[91,1] = PR[90,1] + -30.038;
   1:  PR[91,2] = PR[90,2] + 13.158;
   1:  PR[91,3] = PR[90,3] + 18.183;
   1:L PR[91] R[100]mm/sec CNT100;
   1:  PR[91,1] = PR[90,1] + -30.657;
   1:  PR[91,2] = PR[90,2] + 12.585;
   1:  PR[91,3] = PR[90,3] + 18.189;
   1:L PR[91] R[100]mm/sec CNT100;
   1:  PR[91,1] = PR[90,1] + -31.249;
   1:  PR[91,2] = PR[90,2] + 11.980;
   1:  PR[91,3] = PR[90,3] + 18.195;
   1:L PR[91] R[100]mm/sec CNT100;
   1:  PR[91,1] = PR[90,1] + -31.812;
   1:  PR[91,2] = PR[90,2] + 11.345;
   1:  PR[91,3] = PR[90,3] + 18.200;
   1:L PR[91] R[100]mm/sec CNT100;
   1:  PR[91,1] = PR[90,1] + -32.348;
   1:  PR[91,2] = PR[90,2] + 10.674;
   1:  PR[91,3] = PR[90,3] + 18.206;
   1:L PR[91] R[100]mm/sec CNT100;
   1:  PR[91,1] = PR[90,1] + -32.849;
   1:  PR[91,2] = PR[90,2] + 9.976;
   1:  PR[91,3] = PR[90,3] + 18.212;
   1:L PR[91] R[100]mm/sec CNT100;
   1:  PR[91,1] = PR[90,1] + -33.314;
   1:  PR[91,2] = PR[90,2] + 9.255;
   1:  PR[91,3] = PR[90,3] + 18.218;
   1:L PR[91] R[100]mm/sec CNT100;
   1:  PR[91,1] = PR[90,1] + -33.742;
   1:  PR[91,2] = PR[90,2] + 8.513;
   1:  PR[91,3] = PR[90,3] + 18.224;
   1:L PR[91] R[100]mm/sec CNT100;
   1:  PR[91,1] = PR[90,1] + -34.132;
   1:  PR[91,2] = PR[90,2] + 7.754;
   1:  PR[91,3] = PR[90,3] + 18.230;
   1:L PR[91] R[100]mm/sec CNT100;
   1:  PR[91,1] = PR[90,1] + -34.484;
   1:  PR[91,2] = PR[90,2] + 6.982;
   1:  PR[91,3] = PR[90,3] + 18.236;
   1:L PR[91] R[100]mm/sec CNT100;
   1:  PR[91,1] = PR[90,1] + -34.795;
   1:  PR[91,2] = PR[90,2] + 6.201;
   1:  PR[91,3] = PR[90,3] + 18.241;
   1:L PR[91] R[100]mm/sec CNT100;
   1:  PR[91,1] = PR[90,1] + -35.067;
   1:  PR[91,2] = PR[90,2] + 5.412;
   1:  PR[91,3] = PR[90,3] + 18.247;
   1:L PR[91] R[100]mm/sec CNT100;
   1:  PR[91,1] = PR[90,1] + -35.297;
   1:  PR[91,2] = PR[90,2] + 4.616;
   1:  PR[91,3] = PR[90,3] + 18.253;
   1:L PR[91] R[100]mm/sec CNT100;
   1:  PR[91,1] = PR[90,1] + -35.485;
   1:  PR[91,2] = PR[90,2] + 3.811;
   1:  PR[91,3] = PR[90,3] + 18.259;
   1:L PR[91] R[100]mm/sec CNT100;
   1:  PR[91,1] = PR[90,1] + -35.632;
   1:  PR[91,2] = PR[90,2] + 2.994;
   1:  PR[91,3] = PR[90,3] + 18.264;
   1:L PR[91] R[100]mm/sec CNT100;
   1:  PR[91,1] = PR[90,1] + -35.738;
   1:  PR[91,2] = PR[90,2] + 2.161;
   1:  PR[91,3] = PR[90,3] + 18.270;
   1:L PR[91] R[100]mm/sec CNT100;
   1:  PR[91,1] = PR[90,1] + -35.801;
   1:  PR[91,2] = PR[90,2] + 1.306;
   1:  PR[91,3] = PR[90,3] + 18.276;
   1:L PR[91] R[100]mm/sec CNT100;
   1:  PR[91,1] = PR[90,1] + -35.823;
   1:  PR[91,2] = PR[90,2] + 0.428;
   1:  PR[91,3] = PR[90,3] + 18.281;
   1:L PR[91] R[100]mm/sec CNT100;
   1:  PR[91,1] = PR[90,1] + -35.801;
   1:  PR[91,2] = PR[90,2] + -0.451;
   1:  PR[91,3] = PR[90,3] + 18.288;
   1:L PR[91] R[100]mm/sec CNT100;
   1:  PR[91,1] = PR[90,1] + -35.738;
   1:  PR[91,2] = PR[90,2] + -1.306;
   1:  PR[91,3] = PR[90,3] + 18.294;
   1:L PR[91] R[100]mm/sec CNT100;
   1:  PR[91,1] = PR[90,1] + -35.632;
   1:  PR[91,2] = PR[90,2] + -2.139;
   1:  PR[91,3] = PR[90,3] + 18.299;
   1:L PR[91] R[100]mm/sec CNT100;
   1:  PR[91,1] = PR[90,1] + -35.485;
   1:  PR[91,2] = PR[90,2] + -2.956;
   1:  PR[91,3] = PR[90,3] + 18.305;
   1:L PR[91] R[100]mm/sec CNT100;
   1:  PR[91,1] = PR[90,1] + -35.297;
   1:  PR[91,2] = PR[90,2] + -3.760;
   1:  PR[91,3] = PR[90,3] + 18.311;
   1:L PR[91] R[100]mm/sec CNT100;
   1:  PR[91,1] = PR[90,1] + -35.067;
   1:  PR[91,2] = PR[90,2] + -4.556;
   1:  PR[91,3] = PR[90,3] + 18.317;
   1:L PR[91] R[100]mm/sec CNT100;
   1:  PR[91,1] = PR[90,1] + -34.795;
   1:  PR[91,2] = PR[90,2] + -5.346;
   1:  PR[91,3] = PR[90,3] + 18.322;
   1:L PR[91] R[100]mm/sec CNT100;
   1:  PR[91,1] = PR[90,1] + -34.484;
   1:  PR[91,2] = PR[90,2] + -6.127;
   1:  PR[91,3] = PR[90,3] + 18.328;
   1:L PR[91] R[100]mm/sec CNT100;
   1:  PR[91,1] = PR[90,1] + -34.132;
   1:  PR[91,2] = PR[90,2] + -6.899;
   1:  PR[91,3] = PR[90,3] + 18.334;
   1:L PR[91] R[100]mm/sec CNT100;
   1:  PR[91,1] = PR[90,1] + -33.742;
   1:  PR[91,2] = PR[90,2] + -7.658;
   1:  PR[91,3] = PR[90,3] + 18.340;
   1:L PR[91] R[100]mm/sec CNT100;
   1:  PR[91,1] = PR[90,1] + -33.314;
   1:  PR[91,2] = PR[90,2] + -8.400;
   1:  PR[91,3] = PR[90,3] + 18.345;
   1:L PR[91] R[100]mm/sec CNT100;
   1:  PR[91,1] = PR[90,1] + -32.849;
   1:  PR[91,2] = PR[90,2] + -9.121;
   1:  PR[91,3] = PR[90,3] + 18.351;
   1:L PR[91] R[100]mm/sec CNT100;
   1:  PR[91,1] = PR[90,1] + -32.348;
   1:  PR[91,2] = PR[90,2] + -9.819;
   1:  PR[91,3] = PR[90,3] + 18.357;
   1:L PR[91] R[100]mm/sec CNT100;
   1:  PR[91,1] = PR[90,1] + -31.805;
   1:  PR[91,2] = PR[90,2] + -10.497;
   1:  PR[91,3] = PR[90,3] + 18.363;
   1:L PR[91] R[100]mm/sec CNT100;
   1:  PR[91,1] = PR[90,1] + -31.249;
   1:  PR[91,2] = PR[90,2] + -11.125;
   1:  PR[91,3] = PR[90,3] + 18.369;
   1:L PR[91] R[100]mm/sec CNT100;
   1:  PR[91,1] = PR[90,1] + -30.657;
   1:  PR[91,2] = PR[90,2] + -11.729;
   1:  PR[91,3] = PR[90,3] + 18.375;
   1:L PR[91] R[100]mm/sec CNT100;
   1:  PR[91,1] = PR[90,1] + -30.038;
   1:  PR[91,2] = PR[90,2] + -12.303;
   1:  PR[91,3] = PR[90,3] + 18.380;
   1:L PR[91] R[100]mm/sec CNT100;
   1:  PR[91,1] = PR[90,1] + -29.392;
   1:  PR[91,2] = PR[90,2] + -12.846;
   1:  PR[91,3] = PR[90,3] + 18.386;
   1:L PR[91] R[100]mm/sec CNT100;
   1:  PR[91,1] = PR[90,1] + -28.720;
   1:  PR[91,2] = PR[90,2] + -13.359;
   1:  PR[91,3] = PR[90,3] + 18.392;
   1:L PR[91] R[100]mm/sec CNT100;
   1:  PR[91,1] = PR[90,1] + -28.432;
   1:  PR[91,2] = PR[90,2] + -13.560;
   1:  PR[91,3] = PR[90,3] + 18.398;
   1:L PR[91] R[100]mm/sec CNT100;
   1:  PR[91,1] = PR[90,1] + -28.030;
   1:  PR[91,2] = PR[90,2] + -13.835;
   1:  PR[91,3] = PR[90,3] + 18.400;
   1:L PR[91] R[100]mm/sec CNT100;
   1:  PR[91,1] = PR[90,1] + -27.315;
   1:  PR[91,2] = PR[90,2] + -14.281;
   1:  PR[91,3] = PR[90,3] + 18.404;
   1:L PR[91] R[100]mm/sec CNT100;
   1:  PR[91,1] = PR[90,1] + -26.583;
   1:  PR[91,2] = PR[90,2] + -14.692;
   1:  PR[91,3] = PR[90,3] + 18.409;
   1:L PR[91] R[100]mm/sec CNT100;
   1:  PR[91,1] = PR[90,1] + -25.834;
   1:  PR[91,2] = PR[90,2] + -15.068;
   1:  PR[91,3] = PR[90,3] + 18.415;
   1:L PR[91] R[100]mm/sec CNT100;
   1:  PR[91,1] = PR[90,1] + -25.070;
   1:  PR[91,2] = PR[90,2] + -15.409;
   1:  PR[91,3] = PR[90,3] + 18.421;
   1:L PR[91] R[100]mm/sec CNT100;
   1:  PR[91,1] = PR[90,1] + -24.293;
   1:  PR[91,2] = PR[90,2] + -15.714;
   1:  PR[91,3] = PR[90,3] + 18.427;
   1:L PR[91] R[100]mm/sec CNT100;
   1:  PR[91,1] = PR[90,1] + -23.454;
   1:  PR[91,2] = PR[90,2] + -15.998;
   1:  PR[91,3] = PR[90,3] + 18.432;
   1:L PR[91] R[100]mm/sec CNT100;
   1:  PR[91,1] = PR[90,1] + -22.803;
   1:  PR[91,2] = PR[90,2] + -16.185;
   1:  PR[91,3] = PR[90,3] + 18.438;
   1:L PR[91] R[100]mm/sec CNT100;
   1:  PR[91,1] = PR[90,1] + -21.731;
   1:  PR[91,2] = PR[90,2] + -16.445;
   1:  PR[91,3] = PR[90,3] + 18.443;
   1:L PR[91] R[100]mm/sec CNT100;
   1:  PR[91,1] = PR[90,1] + -20.856;
   1:  PR[91,2] = PR[90,2] + -16.607;
   1:  PR[91,3] = PR[90,3] + 18.451;
   1:L PR[91] R[100]mm/sec CNT100;
   1:  PR[91,1] = PR[90,1] + -19.715;
   1:  PR[91,2] = PR[90,2] + -16.750;
   1:  PR[91,3] = PR[90,3] + 18.457;
   1:L PR[91] R[100]mm/sec CNT100;
   1:  PR[91,1] = PR[90,1] + -19.067;
   1:  PR[91,2] = PR[90,2] + -16.805;
   1:  PR[91,3] = PR[90,3] + 18.465;
   1:L PR[91] R[100]mm/sec CNT100;
   1:  PR[91,1] = PR[90,1] + -18.158;
   1:  PR[91,2] = PR[90,2] + -16.840;
   1:  PR[91,3] = PR[90,3] + 18.469;
   1:L PR[91] R[100]mm/sec CNT100;
   1:  PR[91,1] = PR[90,1] + -17.248;
   1:  PR[91,2] = PR[90,2] + -16.832;
   1:  PR[91,3] = PR[90,3] + 18.475;
   1:L PR[91] R[100]mm/sec CNT100;
   1:  PR[91,1] = PR[90,1] + -16.592;
   1:  PR[91,2] = PR[90,2] + -16.797;
   1:  PR[91,3] = PR[90,3] + 18.482;
   1:L PR[91] R[100]mm/sec CNT100;
   1:  PR[91,1] = PR[90,1] + -15.421;
   1:  PR[91,2] = PR[90,2] + -16.684;
   1:  PR[91,3] = PR[90,3] + 18.486;
   1:L PR[91] R[100]mm/sec CNT100;
   1:  PR[91,1] = PR[90,1] + -14.250;
   1:  PR[91,2] = PR[90,2] + -16.492;
   1:  PR[91,3] = PR[90,3] + 18.494;
   1:L PR[91] R[100]mm/sec CNT100;
   1:  PR[91,1] = PR[90,1] + -13.606;
   1:  PR[91,2] = PR[90,2] + -16.358;
   1:  PR[91,3] = PR[90,3] + 18.502;
   1:L PR[91] R[100]mm/sec CNT100;
   1:  PR[91,1] = PR[90,1] + -12.701;
   1:  PR[91,2] = PR[90,2] + -16.126;
   1:  PR[91,3] = PR[90,3] + 18.507;
   1:L PR[91] R[100]mm/sec CNT100;
   1:  PR[91,1] = PR[90,1] + -11.760;
   1:  PR[91,2] = PR[90,2] + -15.834;
   1:  PR[91,3] = PR[90,3] + 18.513;
   1:L PR[91] R[100]mm/sec CNT100;
   1:  PR[91,1] = PR[90,1] + -11.165;
   1:  PR[91,2] = PR[90,2] + -15.620;
   1:  PR[91,3] = PR[90,3] + 18.520;
   1:L PR[91] R[100]mm/sec CNT100;
   1:  PR[91,1] = PR[90,1] + -10.408;
   1:  PR[91,2] = PR[90,2] + -15.316;
   1:  PR[91,3] = PR[90,3] + 18.524;
   1:L PR[91] R[100]mm/sec CNT100;
   1:  PR[91,1] = PR[90,1] + -9.668;
   1:  PR[91,2] = PR[90,2] + -14.982;
   1:  PR[91,3] = PR[90,3] + 18.530;
   1:L PR[91] R[100]mm/sec CNT100;
   1:  PR[91,1] = PR[90,1] + -9.089;
   1:  PR[91,2] = PR[90,2] + -14.693;
   1:  PR[91,3] = PR[90,3] + 18.535;
   1:L PR[91] R[100]mm/sec CNT100;
   1:  PR[91,1] = PR[90,1] + -8.250;
   1:  PR[91,2] = PR[90,2] + -14.228;
   1:  PR[91,3] = PR[90,3] + 18.540;
   1:L PR[91] R[100]mm/sec CNT100;
   1:  PR[91,1] = PR[90,1] + -7.464;
   1:  PR[91,2] = PR[90,2] + -13.742;
   1:  PR[91,3] = PR[90,3] + 18.546;
   1:L PR[91] R[100]mm/sec CNT100;
   1:  PR[91,1] = PR[90,1] + -6.703;
   1:  PR[91,2] = PR[90,2] + -13.216;
   1:  PR[91,3] = PR[90,3] + 18.553;
   1:L PR[91] R[100]mm/sec CNT100;
   1:  PR[91,1] = PR[90,1] + -6.316;
   1:  PR[91,2] = PR[90,2] + -12.923;
   1:  PR[91,3] = PR[90,3] + 18.559;
   1:L PR[91] R[100]mm/sec CNT100;
   1:  PR[91,1] = PR[90,1] + -5.975;
   1:  PR[91,2] = PR[90,2] + -12.658;
   1:  PR[91,3] = PR[90,3] + 18.562;
   1:L PR[91] R[100]mm/sec CNT100;
   1:  PR[91,1] = PR[90,1] + -5.273;
   1:  PR[91,2] = PR[90,2] + -12.059;
   1:  PR[91,3] = PR[90,3] + 18.565;
   1:L PR[91] R[100]mm/sec CNT100;
   1:  PR[91,1] = PR[90,1] + -4.606;
   1:  PR[91,2] = PR[90,2] + -11.428;
   1:  PR[91,3] = PR[90,3] + 18.572;
   1:L PR[91] R[100]mm/sec CNT100;
   1:  PR[91,1] = PR[90,1] + -3.975;
   1:  PR[91,2] = PR[90,2] + -10.765;
   1:  PR[91,3] = PR[90,3] + 18.578;
   1:L PR[91] R[100]mm/sec CNT100;
   1:  PR[91,1] = PR[90,1] + -3.424;
   1:  PR[91,2] = PR[90,2] + -10.126;
   1:  PR[91,3] = PR[90,3] + 18.584;
   1:L PR[91] R[100]mm/sec CNT100;
   1:  PR[91,1] = PR[90,1] + -2.950;
   1:  PR[91,2] = PR[90,2] + -9.517;
   1:  PR[91,3] = PR[90,3] + 18.590;
   1:L PR[91] R[100]mm/sec CNT100;
   1:  PR[91,1] = PR[90,1] + -2.338;
   1:  PR[91,2] = PR[90,2] + -8.667;
   1:  PR[91,3] = PR[90,3] + 18.595;
   1:L PR[91] R[100]mm/sec CNT100;
   1:  PR[91,1] = PR[90,1] + -2.051;
   1:  PR[91,2] = PR[90,2] + -8.363;
   1:  PR[91,3] = PR[90,3] + 18.602;
   1:L PR[91] R[100]mm/sec CNT100;
   1:  PR[91,1] = PR[90,1] + -1.719;
   1:  PR[91,2] = PR[90,2] + -8.092;
   1:  PR[91,3] = PR[90,3] + 18.605;
   1:L PR[91] R[100]mm/sec CNT100;
   1:  PR[91,1] = PR[90,1] + -1.330;
   1:  PR[91,2] = PR[90,2] + -7.859;
   1:  PR[91,3] = PR[90,3] + 18.608;
   1:L PR[91] R[100]mm/sec CNT100;
   1:  PR[91,1] = PR[90,1] + -0.898;
   1:  PR[91,2] = PR[90,2] + -7.690;
   1:  PR[91,3] = PR[90,3] + 18.611;
   1:L PR[91] R[100]mm/sec CNT100;
   1:  PR[91,1] = PR[90,1] + -0.547;
   1:  PR[91,2] = PR[90,2] + -7.606;
   1:  PR[91,3] = PR[90,3] + 18.615;
   1:L PR[91] R[100]mm/sec CNT100;
   1:  PR[91,1] = PR[90,1] + -0.119;
   1:  PR[91,2] = PR[90,2] + -7.571;
   1:  PR[91,3] = PR[90,3] + 18.617;
   1:L PR[91] R[100]mm/sec CNT100;
   1:  PR[91] = PR[90];
   1:  PR[91,1] = PR[90,1] + 0.183;
   1:  PR[91,2] = PR[90,2] + -8.483;
   1:  PR[91,3] = PR[90,3] + 19.950;
   1:L PR[91] R[100]mm/sec CNT100;
   1:  PR[91,1] = PR[90,1] + 0.672;
   1:  PR[91,2] = PR[90,2] + -8.583;
   1:  PR[91,3] = PR[90,3] + 18.621;
   1:L PR[91] R[100]mm/sec CNT100;
   1:  PR[91,1] = PR[90,1] + 1.149;
   1:  PR[91,2] = PR[90,2] + -8.776;
   1:  PR[91,3] = PR[90,3] + 18.625;
   1:L PR[91] R[100]mm/sec CNT100;
   1:  PR[91,1] = PR[90,1] + 1.590;
   1:  PR[91,2] = PR[90,2] + -9.054;
   1:  PR[91,3] = PR[90,3] + 18.629;
   1:L PR[91] R[100]mm/sec CNT100;
   1:  PR[91,1] = PR[90,1] + 1.985;
   1:  PR[91,2] = PR[90,2] + -9.410;
   1:  PR[91,3] = PR[90,3] + 18.632;
   1:L PR[91] R[100]mm/sec CNT100;
   1:  PR[91,1] = PR[90,1] + 2.709;
   1:  PR[91,2] = PR[90,2] + -10.314;
   1:  PR[91,3] = PR[90,3] + 18.636;
   1:L PR[91] R[100]mm/sec CNT100;
   1:  PR[91,1] = PR[90,1] + 3.083;
   1:  PR[91,2] = PR[90,2] + -10.749;
   1:  PR[91,3] = PR[90,3] + 18.644;
   1:L PR[91] R[100]mm/sec CNT100;
   1:  PR[91,1] = PR[90,1] + 3.538;
   1:  PR[91,2] = PR[90,2] + -11.238;
   1:  PR[91,3] = PR[90,3] + 18.648;
   1:L PR[91] R[100]mm/sec CNT100;
   1:  PR[91,1] = PR[90,1] + 3.917;
   1:  PR[91,2] = PR[90,2] + -11.619;
   1:  PR[91,3] = PR[90,3] + 18.653;
   1:L PR[91] R[100]mm/sec CNT100;
   1:  PR[91,1] = PR[90,1] + 4.391;
   1:  PR[91,2] = PR[90,2] + -12.065;
   1:  PR[91,3] = PR[90,3] + 18.656;
   1:L PR[91] R[100]mm/sec CNT100;
   1:  PR[91,1] = PR[90,1] + 4.857;
   1:  PR[91,2] = PR[90,2] + -12.470;
   1:  PR[91,3] = PR[90,3] + 18.661;
   1:L PR[91] R[100]mm/sec CNT100;
   1:  PR[91,1] = PR[90,1] + 5.822;
   1:  PR[91,2] = PR[90,2] + -13.229;
   1:  PR[91,3] = PR[90,3] + 18.665;
   1:L PR[91] R[100]mm/sec CNT100;
   1:  PR[91,1] = PR[90,1] + 6.732;
   1:  PR[91,2] = PR[90,2] + -13.853;
   1:  PR[91,3] = PR[90,3] + 18.674;
   1:L PR[91] R[100]mm/sec CNT100;
   1:  PR[91,1] = PR[90,1] + 7.341;
   1:  PR[91,2] = PR[90,2] + -14.231;
   1:  PR[91,3] = PR[90,3] + 18.681;
   1:L PR[91] R[100]mm/sec CNT100;
   1:  PR[91,1] = PR[90,1] + 8.044;
   1:  PR[91,2] = PR[90,2] + -14.626;
   1:  PR[91,3] = PR[90,3] + 18.686;
   1:L PR[91] R[100]mm/sec CNT100;
   1:  PR[91,1] = PR[90,1] + 8.891;
   1:  PR[91,2] = PR[90,2] + -15.051;
   1:  PR[91,3] = PR[90,3] + 18.692;
   1:L PR[91] R[100]mm/sec CNT100;
   1:  PR[91,1] = PR[90,1] + 9.732;
   1:  PR[91,2] = PR[90,2] + -15.426;
   1:  PR[91,3] = PR[90,3] + 18.698;
   1:L PR[91] R[100]mm/sec CNT100;
   1:  PR[91,1] = PR[90,1] + 10.607;
   1:  PR[91,2] = PR[90,2] + -15.766;
   1:  PR[91,3] = PR[90,3] + 18.705;
   1:L PR[91] R[100]mm/sec CNT100;
   1:  PR[91,1] = PR[90,1] + 11.072;
   1:  PR[91,2] = PR[90,2] + -15.924;
   1:  PR[91,3] = PR[90,3] + 18.711;
   1:L PR[91] R[100]mm/sec CNT100;
   1:  PR[91,1] = PR[90,1] + 11.492;
   1:  PR[91,2] = PR[90,2] + -16.062;
   1:  PR[91,3] = PR[90,3] + 18.715;
   1:L PR[91] R[100]mm/sec CNT100;
   1:  PR[91,1] = PR[90,1] + 12.394;
   1:  PR[91,2] = PR[90,2] + -16.315;
   1:  PR[91,3] = PR[90,3] + 18.718;
   1:L PR[91] R[100]mm/sec CNT100;
   1:  PR[91,1] = PR[90,1] + 13.326;
   1:  PR[91,2] = PR[90,2] + -16.529;
   1:  PR[91,3] = PR[90,3] + 18.724;
   1:L PR[91] R[100]mm/sec CNT100;
   1:  PR[91,1] = PR[90,1] + 14.124;
   1:  PR[91,2] = PR[90,2] + -16.675;
   1:  PR[91,3] = PR[90,3] + 18.731;
   1:L PR[91] R[100]mm/sec CNT100;
   1:  PR[91,1] = PR[90,1] + 14.940;
   1:  PR[91,2] = PR[90,2] + -16.788;
   1:  PR[91,3] = PR[90,3] + 18.737;
   1:L PR[91] R[100]mm/sec CNT100;
   1:  PR[91,1] = PR[90,1] + 15.766;
   1:  PR[91,2] = PR[90,2] + -16.867;
   1:  PR[91,3] = PR[90,3] + 18.742;
   1:L PR[91] R[100]mm/sec CNT100;
   1:  PR[91,1] = PR[90,1] + 16.242;
   1:  PR[91,2] = PR[90,2] + -16.895;
   1:  PR[91,3] = PR[90,3] + 18.748;
   1:L PR[91] R[100]mm/sec CNT100;
   1:  PR[91,1] = PR[90,1] + 17.434;
   1:  PR[91,2] = PR[90,2] + -16.918;
   1:  PR[91,3] = PR[90,3] + 18.751;
   1:L PR[91] R[100]mm/sec CNT100;
   1:  PR[91,1] = PR[90,1] + 18.271;
   1:  PR[91,2] = PR[90,2] + -16.889;
   1:  PR[91,3] = PR[90,3] + 18.760;
   1:L PR[91] R[100]mm/sec CNT100;
   1:  PR[91,1] = PR[90,1] + 19.174;
   1:  PR[91,2] = PR[90,2] + -16.818;
   1:  PR[91,3] = PR[90,3] + 18.766;
   1:L PR[91] R[100]mm/sec CNT100;
   1:  PR[91,1] = PR[90,1] + 20.083;
   1:  PR[91,2] = PR[90,2] + -16.702;
   1:  PR[91,3] = PR[90,3] + 18.772;
   1:L PR[91] R[100]mm/sec CNT100;
   1:  PR[91,1] = PR[90,1] + 20.980;
   1:  PR[91,2] = PR[90,2] + -16.543;
   1:  PR[91,3] = PR[90,3] + 18.778;
   1:L PR[91] R[100]mm/sec CNT100;
   1:  PR[91,1] = PR[90,1] + 21.866;
   1:  PR[91,2] = PR[90,2] + -16.341;
   1:  PR[91,3] = PR[90,3] + 18.785;
   1:L PR[91] R[100]mm/sec CNT100;
   1:  PR[91,1] = PR[90,1] + 22.738;
   1:  PR[91,2] = PR[90,2] + -16.098;
   1:  PR[91,3] = PR[90,3] + 18.791;
   1:L PR[91] R[100]mm/sec CNT100;
   1:  PR[91,1] = PR[90,1] + 23.593;
   1:  PR[91,2] = PR[90,2] + -15.816;
   1:  PR[91,3] = PR[90,3] + 18.797;
   1:L PR[91] R[100]mm/sec CNT100;
   1:  PR[91,1] = PR[90,1] + 24.429;
   1:  PR[91,2] = PR[90,2] + -15.494;
   1:  PR[91,3] = PR[90,3] + 18.803;
   1:L PR[91] R[100]mm/sec CNT100;
   1:  PR[91,1] = PR[90,1] + 25.241;
   1:  PR[91,2] = PR[90,2] + -15.136;
   1:  PR[91,3] = PR[90,3] + 18.810;
   1:L PR[91] R[100]mm/sec CNT100;
   1:  PR[91,1] = PR[90,1] + 26.032;
   1:  PR[91,2] = PR[90,2] + -14.741;
   1:  PR[91,3] = PR[90,3] + 18.816;
   1:L PR[91] R[100]mm/sec CNT100;
   1:  PR[91,1] = PR[90,1] + 26.799;
   1:  PR[91,2] = PR[90,2] + -14.311;
   1:  PR[91,3] = PR[90,3] + 18.822;
   1:L PR[91] R[100]mm/sec CNT100;
   1:  PR[91,1] = PR[90,1] + 27.542;
   1:  PR[91,2] = PR[90,2] + -13.847;
   1:  PR[91,3] = PR[90,3] + 18.828;
   1:L PR[91] R[100]mm/sec CNT100;
   1:  PR[91,1] = PR[90,1] + 28.258;
   1:  PR[91,2] = PR[90,2] + -13.349;
   1:  PR[91,3] = PR[90,3] + 18.834;
   1:L PR[91] R[100]mm/sec CNT100;
   1:  PR[91,1] = PR[90,1] + 28.946;
   1:  PR[91,2] = PR[90,2] + -12.819;
   1:  PR[91,3] = PR[90,3] + 18.840;
   1:L PR[91] R[100]mm/sec CNT100;
   1:  PR[91,1] = PR[90,1] + 29.606;
   1:  PR[91,2] = PR[90,2] + -12.258;
   1:  PR[91,3] = PR[90,3] + 18.846;
   1:L PR[91] R[100]mm/sec CNT100;
   1:  PR[91,1] = PR[90,1] + 30.234;
   1:  PR[91,2] = PR[90,2] + -11.667;
   1:  PR[91,3] = PR[90,3] + 18.852;
   1:L PR[91] R[100]mm/sec CNT100;
   1:  PR[91,1] = PR[90,1] + 30.841;
   1:  PR[91,2] = PR[90,2] + -11.036;
   1:  PR[91,3] = PR[90,3] + 18.858;
   1:L PR[91] R[100]mm/sec CNT100;
   1:  PR[91,1] = PR[90,1] + 31.384;
   1:  PR[91,2] = PR[90,2] + -10.410;
   1:  PR[91,3] = PR[90,3] + 18.864;
   1:L PR[91] R[100]mm/sec CNT100;
   1:  PR[91,1] = PR[90,1] + 31.905;
   1:  PR[91,2] = PR[90,2] + -9.747;
   1:  PR[91,3] = PR[90,3] + 18.870;
   1:L PR[91] R[100]mm/sec CNT100;
   1:  PR[91,1] = PR[90,1] + 32.393;
   1:  PR[91,2] = PR[90,2] + -9.059;
   1:  PR[91,3] = PR[90,3] + 18.876;
   1:L PR[91] R[100]mm/sec CNT100;
   1:  PR[91,1] = PR[90,1] + 32.848;
   1:  PR[91,2] = PR[90,2] + -8.348;
   1:  PR[91,3] = PR[90,3] + 18.882;
   1:L PR[91] R[100]mm/sec CNT100;
   1:  PR[91,1] = PR[90,1] + 33.269;
   1:  PR[91,2] = PR[90,2] + -7.617;
   1:  PR[91,3] = PR[90,3] + 18.888;
   1:L PR[91] R[100]mm/sec CNT100;
   1:  PR[91,1] = PR[90,1] + 33.653;
   1:  PR[91,2] = PR[90,2] + -6.869;
   1:  PR[91,3] = PR[90,3] + 18.894;
   1:L PR[91] R[100]mm/sec CNT100;
   1:  PR[91,1] = PR[90,1] + 34.001;
   1:  PR[91,2] = PR[90,2] + -6.109;
   1:  PR[91,3] = PR[90,3] + 18.899;
   1:L PR[91] R[100]mm/sec CNT100;
   1:  PR[91,1] = PR[90,1] + 34.309;
   1:  PR[91,2] = PR[90,2] + -5.339;
   1:  PR[91,3] = PR[90,3] + 18.905;
   1:L PR[91] R[100]mm/sec CNT100;
   1:  PR[91,1] = PR[90,1] + 34.578;
   1:  PR[91,2] = PR[90,2] + -4.560;
   1:  PR[91,3] = PR[90,3] + 18.911;
   1:L PR[91] R[100]mm/sec CNT100;
   1:  PR[91,1] = PR[90,1] + 34.807;
   1:  PR[91,2] = PR[90,2] + -3.771;
   1:  PR[91,3] = PR[90,3] + 18.917;
   1:L PR[91] R[100]mm/sec CNT100;
   1:  PR[91,1] = PR[90,1] + 34.995;
   1:  PR[91,2] = PR[90,2] + -2.969;
   1:  PR[91,3] = PR[90,3] + 18.922;
   1:L PR[91] R[100]mm/sec CNT100;
   1:  PR[91,1] = PR[90,1] + 35.142;
   1:  PR[91,2] = PR[90,2] + -2.152;
   1:  PR[91,3] = PR[90,3] + 18.928;
   1:L PR[91] R[100]mm/sec CNT100;
   1:  PR[91,1] = PR[90,1] + 35.247;
   1:  PR[91,2] = PR[90,2] + -1.316;
   1:  PR[91,3] = PR[90,3] + 18.934;
   1:L PR[91] R[100]mm/sec CNT100;
   1:  PR[91,1] = PR[90,1] + 35.311;
   1:  PR[91,2] = PR[90,2] + -0.457;
   1:  PR[91,3] = PR[90,3] + 18.940;
   1:L PR[91] R[100]mm/sec CNT100;
   1:  PR[91,1] = PR[90,1] + 35.332;
   1:  PR[91,2] = PR[90,2] + 0.428;
   1:  PR[91,3] = PR[90,3] + 18.946;
   1:L PR[91] R[100]mm/sec CNT100;
   1:  PR[91,1] = PR[90,1] + 35.311;
   1:  PR[91,2] = PR[90,2] + 1.312;
   1:  PR[91,3] = PR[90,3] + 18.952;
   1:L PR[91] R[100]mm/sec CNT100;
   1:  PR[91,1] = PR[90,1] + 35.247;
   1:  PR[91,2] = PR[90,2] + 2.171;
   1:  PR[91,3] = PR[90,3] + 18.958;
   1:L PR[91] R[100]mm/sec CNT100;
   1:  PR[91,1] = PR[90,1] + 35.142;
   1:  PR[91,2] = PR[90,2] + 3.007;
   1:  PR[91,3] = PR[90,3] + 18.964;
   1:L PR[91] R[100]mm/sec CNT100;
   1:  PR[91,1] = PR[90,1] + 34.995;
   1:  PR[91,2] = PR[90,2] + 3.824;
   1:  PR[91,3] = PR[90,3] + 18.970;
   1:L PR[91] R[100]mm/sec CNT100;
   1:  PR[91,1] = PR[90,1] + 34.807;
   1:  PR[91,2] = PR[90,2] + 4.626;
   1:  PR[91,3] = PR[90,3] + 18.976;
   1:L PR[91] R[100]mm/sec CNT100;
   1:  PR[91,1] = PR[90,1] + 34.578;
   1:  PR[91,2] = PR[90,2] + 5.415;
   1:  PR[91,3] = PR[90,3] + 18.981;
   1:L PR[91] R[100]mm/sec CNT100;
   1:  PR[91,1] = PR[90,1] + 34.309;
   1:  PR[91,2] = PR[90,2] + 6.194;
   1:  PR[91,3] = PR[90,3] + 18.987;
   1:L PR[91] R[100]mm/sec CNT100;
   1:  PR[91,1] = PR[90,1] + 34.001;
   1:  PR[91,2] = PR[90,2] + 6.964;
   1:  PR[91,3] = PR[90,3] + 18.993;
   1:L PR[91] R[100]mm/sec CNT100;
   1:  PR[91,1] = PR[90,1] + 33.653;
   1:  PR[91,2] = PR[90,2] + 7.724;
   1:  PR[91,3] = PR[90,3] + 18.999;
   1:L PR[91] R[100]mm/sec CNT100;
   1:  PR[91,1] = PR[90,1] + 33.269;
   1:  PR[91,2] = PR[90,2] + 8.472;
   1:  PR[91,3] = PR[90,3] + 19.004;
   1:L PR[91] R[100]mm/sec CNT100;
   1:  PR[91,1] = PR[90,1] + 32.963;
   1:  PR[91,2] = PR[90,2] + 9.006;
   1:  PR[91,3] = PR[90,3] + 19.010;
   1:L PR[91] R[100]mm/sec CNT100;
   1:  PR[91,1] = PR[90,1] + 32.391;
   1:  PR[91,2] = PR[90,2] + 9.916;
   1:  PR[91,3] = PR[90,3] + 19.014;
   1:L PR[91] R[100]mm/sec CNT100;
   1:  PR[91,1] = PR[90,1] + 31.905;
   1:  PR[91,2] = PR[90,2] + 10.602;
   1:  PR[91,3] = PR[90,3] + 19.022;
   1:L PR[91] R[100]mm/sec CNT100;
   1:  PR[91,1] = PR[90,1] + 31.384;
   1:  PR[91,2] = PR[90,2] + 11.265;
   1:  PR[91,3] = PR[90,3] + 19.028;
   1:L PR[91] R[100]mm/sec CNT100;
   1:  PR[91,1] = PR[90,1] + 30.831;
   1:  PR[91,2] = PR[90,2] + 11.902;
   1:  PR[91,3] = PR[90,3] + 19.034;
   1:L PR[91] R[100]mm/sec CNT100;
   1:  PR[91,1] = PR[90,1] + 30.234;
   1:  PR[91,2] = PR[90,2] + 12.522;
   1:  PR[91,3] = PR[90,3] + 19.040;
   1:L PR[91] R[100]mm/sec CNT100;
   1:  PR[91,1] = PR[90,1] + 29.605;
   1:  PR[91,2] = PR[90,2] + 13.113;
   1:  PR[91,3] = PR[90,3] + 19.045;
   1:L PR[91] R[100]mm/sec CNT100;
   1:  PR[91,1] = PR[90,1] + 28.947;
   1:  PR[91,2] = PR[90,2] + 13.674;
   1:  PR[91,3] = PR[90,3] + 19.051;
   1:L PR[91] R[100]mm/sec CNT100;
   1:  PR[91,1] = PR[90,1] + 28.257;
   1:  PR[91,2] = PR[90,2] + 14.204;
   1:  PR[91,3] = PR[90,3] + 19.058;
   1:L PR[91] R[100]mm/sec CNT100;
   1:  PR[91,1] = PR[90,1] + 27.858;
   1:  PR[91,2] = PR[90,2] + 14.484;
   1:  PR[91,3] = PR[90,3] + 19.064;
   1:L PR[91] R[100]mm/sec CNT100;
   1:  PR[91,1] = PR[90,1] + 27.543;
   1:  PR[91,2] = PR[90,2] + 14.701;
   1:  PR[91,3] = PR[90,3] + 19.067;
   1:L PR[91] R[100]mm/sec CNT100;
   1:  PR[91,1] = PR[90,1] + 26.799;
   1:  PR[91,2] = PR[90,2] + 15.167;
   1:  PR[91,3] = PR[90,3] + 19.070;
   1:L PR[91] R[100]mm/sec CNT100;
   1:  PR[91,1] = PR[90,1] + 26.032;
   1:  PR[91,2] = PR[90,2] + 15.597;
   1:  PR[91,3] = PR[90,3] + 19.076;
   1:L PR[91] R[100]mm/sec CNT100;
   1:  PR[91,1] = PR[90,1] + 25.241;
   1:  PR[91,2] = PR[90,2] + 15.991;
   1:  PR[91,3] = PR[90,3] + 19.082;
   1:L PR[91] R[100]mm/sec CNT100;
   1:  PR[91,1] = PR[90,1] + 24.429;
   1:  PR[91,2] = PR[90,2] + 16.349;
   1:  PR[91,3] = PR[90,3] + 19.088;
   1:L PR[91] R[100]mm/sec CNT100;
   1:  PR[91,1] = PR[90,1] + 23.593;
   1:  PR[91,2] = PR[90,2] + 16.671;
   1:  PR[91,3] = PR[90,3] + 19.094;
   1:L PR[91] R[100]mm/sec CNT100;
   1:  PR[91,1] = PR[90,1] + 22.921;
   1:  PR[91,2] = PR[90,2] + 16.894;
   1:  PR[91,3] = PR[90,3] + 19.100;
   1:L PR[91] R[100]mm/sec CNT100;
   1:  PR[91,1] = PR[90,1] + 21.864;
   1:  PR[91,2] = PR[90,2] + 17.197;
   1:  PR[91,3] = PR[90,3] + 19.105;
   1:L PR[91] R[100]mm/sec CNT100;
   1:  PR[91,1] = PR[90,1] + 20.979;
   1:  PR[91,2] = PR[90,2] + 17.398;
   1:  PR[91,3] = PR[90,3] + 19.113;
   1:L PR[91] R[100]mm/sec CNT100;
   1:  PR[91,1] = PR[90,1] + 20.625;
   1:  PR[91,2] = PR[90,2] + 17.462;
   1:  PR[91,3] = PR[90,3] + 19.119;
   1:L PR[91] R[100]mm/sec CNT100;
   1:  PR[91,1] = PR[90,1] + 20.083;
   1:  PR[91,2] = PR[90,2] + 17.557;
   1:  PR[91,3] = PR[90,3] + 19.122;
   1:L PR[91] R[100]mm/sec CNT100;
   1:  PR[91,1] = PR[90,1] + 19.174;
   1:  PR[91,2] = PR[90,2] + 17.673;
   1:  PR[91,3] = PR[90,3] + 19.126;
   1:L PR[91] R[100]mm/sec CNT100;
   1:  PR[91,1] = PR[90,1] + 18.243;
   1:  PR[91,2] = PR[90,2] + 17.746;
   1:  PR[91,3] = PR[90,3] + 19.132;
   1:L PR[91] R[100]mm/sec CNT100;
   1:  PR[91,1] = PR[90,1] + 17.434;
   1:  PR[91,2] = PR[90,2] + 17.773;
   1:  PR[91,3] = PR[90,3] + 19.138;
   1:L PR[91] R[100]mm/sec CNT100;
   1:  PR[91,1] = PR[90,1] + 16.241;
   1:  PR[91,2] = PR[90,2] + 17.751;
   1:  PR[91,3] = PR[90,3] + 19.144;
   1:L PR[91] R[100]mm/sec CNT100;
   1:  PR[91,1] = PR[90,1] + 15.766;
   1:  PR[91,2] = PR[90,2] + 17.722;
   1:  PR[91,3] = PR[90,3] + 19.152;
   1:L PR[91] R[100]mm/sec CNT100;
   1:  PR[91,1] = PR[90,1] + 14.939;
   1:  PR[91,2] = PR[90,2] + 17.643;
   1:  PR[91,3] = PR[90,3] + 19.156;
   1:L PR[91] R[100]mm/sec CNT100;
   1:  PR[91,1] = PR[90,1] + 14.124;
   1:  PR[91,2] = PR[90,2] + 17.530;
   1:  PR[91,3] = PR[90,3] + 19.161;
   1:L PR[91] R[100]mm/sec CNT100;
   1:  PR[91,1] = PR[90,1] + 13.305;
   1:  PR[91,2] = PR[90,2] + 17.380;
   1:  PR[91,3] = PR[90,3] + 19.167;
   1:L PR[91] R[100]mm/sec CNT100;
   1:  PR[91,1] = PR[90,1] + 12.393;
   1:  PR[91,2] = PR[90,2] + 17.170;
   1:  PR[91,3] = PR[90,3] + 19.173;
   1:L PR[91] R[100]mm/sec CNT100;
   1:  PR[91,1] = PR[90,1] + 11.811;
   1:  PR[91,2] = PR[90,2] + 17.009;
   1:  PR[91,3] = PR[90,3] + 19.179;
   1:L PR[91] R[100]mm/sec CNT100;
   1:  PR[91,1] = PR[90,1] + 11.496;
   1:  PR[91,2] = PR[90,2] + 16.918;
   1:  PR[91,3] = PR[90,3] + 19.184;
   1:L PR[91] R[100]mm/sec CNT100;
   1:  PR[91,1] = PR[90,1] + 10.607;
   1:  PR[91,2] = PR[90,2] + 16.621;
   1:  PR[91,3] = PR[90,3] + 19.186;
   1:L PR[91] R[100]mm/sec CNT100;
   1:  PR[91,1] = PR[90,1] + 9.615;
   1:  PR[91,2] = PR[90,2] + 16.230;
   1:  PR[91,3] = PR[90,3] + 19.192;
   1:L PR[91] R[100]mm/sec CNT100;
   1:  PR[91,1] = PR[90,1] + 8.863;
   1:  PR[91,2] = PR[90,2] + 15.893;
   1:  PR[91,3] = PR[90,3] + 19.200;
   1:L PR[91] R[100]mm/sec CNT100;
   1:  PR[91,1] = PR[90,1] + 8.175;
   1:  PR[91,2] = PR[90,2] + 15.549;
   1:  PR[91,3] = PR[90,3] + 19.206;
   1:L PR[91] R[100]mm/sec CNT100;
   1:  PR[91,1] = PR[90,1] + 7.342;
   1:  PR[91,2] = PR[90,2] + 15.086;
   1:  PR[91,3] = PR[90,3] + 19.211;
   1:L PR[91] R[100]mm/sec CNT100;
   1:  PR[91,1] = PR[90,1] + 6.397;
   1:  PR[91,2] = PR[90,2] + 14.489;
   1:  PR[91,3] = PR[90,3] + 19.217;
   1:L PR[91] R[100]mm/sec CNT100;
   1:  PR[91,1] = PR[90,1] + 5.821;
   1:  PR[91,2] = PR[90,2] + 14.083;
   1:  PR[91,3] = PR[90,3] + 19.225;
   1:L PR[91] R[100]mm/sec CNT100;
   1:  PR[91,1] = PR[90,1] + 5.323;
   1:  PR[91,2] = PR[90,2] + 13.704;
   1:  PR[91,3] = PR[90,3] + 19.230;
   1:L PR[91] R[100]mm/sec CNT100;
   1:  PR[91,1] = PR[90,1] + 4.837;
   1:  PR[91,2] = PR[90,2] + 13.309;
   1:  PR[91,3] = PR[90,3] + 19.235;
   1:L PR[91] R[100]mm/sec CNT100;
   1:  PR[91,1] = PR[90,1] + 4.392;
   1:  PR[91,2] = PR[90,2] + 12.920;
   1:  PR[91,3] = PR[90,3] + 19.239;
   1:L PR[91] R[100]mm/sec CNT100;
   1:  PR[91,1] = PR[90,1] + 3.917;
   1:  PR[91,2] = PR[90,2] + 12.474;
   1:  PR[91,3] = PR[90,3] + 19.243;
   1:L PR[91] R[100]mm/sec CNT100;
   1:  PR[91,1] = PR[90,1] + 3.538;
   1:  PR[91,2] = PR[90,2] + 12.093;
   1:  PR[91,3] = PR[90,3] + 19.247;
   1:L PR[91] R[100]mm/sec CNT100;
   1:  PR[91,1] = PR[90,1] + 3.084;
   1:  PR[91,2] = PR[90,2] + 11.605;
   1:  PR[91,3] = PR[90,3] + 19.251;
   1:L PR[91] R[100]mm/sec CNT100;
   1:  PR[91,1] = PR[90,1] + 2.634;
   1:  PR[91,2] = PR[90,2] + 11.077;
   1:  PR[91,3] = PR[90,3] + 19.256;
   1:L PR[91] R[100]mm/sec CNT100;
   1:  PR[91,1] = PR[90,1] + 2.059;
   1:  PR[91,2] = PR[90,2] + 10.347;
   1:  PR[91,3] = PR[90,3] + 19.261;
   1:L PR[91] R[100]mm/sec CNT100;
   1:  PR[91,1] = PR[90,1] + 1.765;
   1:  PR[91,2] = PR[90,2] + 10.056;
   1:  PR[91,3] = PR[90,3] + 19.267;
   1:L PR[91] R[100]mm/sec CNT100;
   1:  PR[91,1] = PR[90,1] + 1.580;
   1:  PR[91,2] = PR[90,2] + 9.903;
   1:  PR[91,3] = PR[90,3] + 19.270;
   1:L PR[91] R[100]mm/sec CNT100;
   1:  PR[91,1] = PR[90,1] + 1.154;
   1:  PR[91,2] = PR[90,2] + 9.635;
   1:  PR[91,3] = PR[90,3] + 19.272;
   1:L PR[91] R[100]mm/sec CNT100;
   1:  PR[91,1] = PR[90,1] + 0.784;
   1:  PR[91,2] = PR[90,2] + 9.475;
   1:  PR[91,3] = PR[90,3] + 19.275;
   1:L PR[91] R[100]mm/sec CNT100;
   1:  PR[91,1] = PR[90,1] + 0.375;
   1:  PR[91,2] = PR[90,2] + 9.366;
   1:  PR[91,3] = PR[90,3] + 19.278;
   1:L PR[91] R[100]mm/sec CNT100;
   1:  PR[91,1] = PR[90,1] + -0.138;
   1:  PR[91,2] = PR[90,2] + 9.320;
   1:  PR[91,3] = PR[90,3] + 19.281;
   1:L PR[91] R[100]mm/sec CNT100;
   1:  PR[91,1] = PR[90,1] + -0.659;
   1:  PR[91,2] = PR[90,2] + 9.376;
   1:  PR[91,3] = PR[90,3] + 19.285;
   1:L PR[91] R[100]mm/sec CNT100;
   1:  PR[91,1] = PR[90,1] + -1.062;
   1:  PR[91,2] = PR[90,2] + 9.492;
   1:  PR[91,3] = PR[90,3] + 19.288;
   1:L PR[91] R[100]mm/sec CNT100;
   1:  PR[91,1] = PR[90,1] + -1.298;
   1:  PR[91,2] = PR[90,2] + 9.591;
   1:  PR[91,3] = PR[90,3] + 19.291;
   1:L PR[91] R[100]mm/sec CNT100;
   1:  PR[91,1] = PR[90,1] + -1.614;
   1:  PR[91,2] = PR[90,2] + 9.764;
   1:  PR[91,3] = PR[90,3] + 19.293;
   1:L PR[91] R[100]mm/sec CNT100;
   1:  PR[91,1] = PR[90,1] + -2.072;
   1:  PR[91,2] = PR[90,2] + 10.117;
   1:  PR[91,3] = PR[90,3] + 19.295;
   1:L PR[91] R[100]mm/sec CNT100;
   1:  PR[91,1] = PR[90,1] + -2.432;
   1:  PR[91,2] = PR[90,2] + 10.528;
   1:  PR[91,3] = PR[90,3] + 19.299;
   1:L PR[91] R[100]mm/sec CNT100;
   1:  PR[91,1] = PR[90,1] + -2.857;
   1:  PR[91,2] = PR[90,2] + 11.068;
   1:  PR[91,3] = PR[90,3] + 19.303;
   1:L PR[91] R[100]mm/sec CNT100;
   1:  PR[91,1] = PR[90,1] + -3.300;
   1:  PR[91,2] = PR[90,2] + 11.586;
   1:  PR[91,3] = PR[90,3] + 19.308;
   1:L PR[91] R[100]mm/sec CNT100;
   1:  PR[91,1] = PR[90,1] + -4.134;
   1:  PR[91,2] = PR[90,2] + 12.455;
   1:  PR[91,3] = PR[90,3] + 19.313;
   1:L PR[91] R[100]mm/sec CNT100;
   1:  PR[91,1] = PR[90,1] + -4.605;
   1:  PR[91,2] = PR[90,2] + 12.897;
   1:  PR[91,3] = PR[90,3] + 19.321;
   1:L PR[91] R[100]mm/sec CNT100;
   1:  PR[91,1] = PR[90,1] + -5.076;
   1:  PR[91,2] = PR[90,2] + 13.307;
   1:  PR[91,3] = PR[90,3] + 19.326;
   1:L PR[91] R[100]mm/sec CNT100;
   1:  PR[91,1] = PR[90,1] + -5.562;
   1:  PR[91,2] = PR[90,2] + 13.702;
   1:  PR[91,3] = PR[90,3] + 19.330;
   1:L PR[91] R[100]mm/sec CNT100;
   1:  PR[91,1] = PR[90,1] + -6.044;
   1:  PR[91,2] = PR[90,2] + 14.068;
   1:  PR[91,3] = PR[90,3] + 19.334;
   1:L PR[91] R[100]mm/sec CNT100;
   1:  PR[91,1] = PR[90,1] + -6.624;
   1:  PR[91,2] = PR[90,2] + 14.477;
   1:  PR[91,3] = PR[90,3] + 19.338;
   1:L PR[91] R[100]mm/sec CNT100;
   1:  PR[91,1] = PR[90,1] + -7.576;
   1:  PR[91,2] = PR[90,2] + 15.080;
   1:  PR[91,3] = PR[90,3] + 19.343;
   1:L PR[91] R[100]mm/sec CNT100;
   1:  PR[91,1] = PR[90,1] + -8.410;
   1:  PR[91,2] = PR[90,2] + 15.546;
   1:  PR[91,3] = PR[90,3] + 19.351;
   1:L PR[91] R[100]mm/sec CNT100;
   1:  PR[91,1] = PR[90,1] + -9.123;
   1:  PR[91,2] = PR[90,2] + 15.903;
   1:  PR[91,3] = PR[90,3] + 19.358;
   1:L PR[91] R[100]mm/sec CNT100;
   1:  PR[91,1] = PR[90,1] + -9.964;
   1:  PR[91,2] = PR[90,2] + 16.279;
   1:  PR[91,3] = PR[90,3] + 19.363;
   1:L PR[91] R[100]mm/sec CNT100;
   1:  PR[91,1] = PR[90,1] + -10.840;
   1:  PR[91,2] = PR[90,2] + 16.621;
   1:  PR[91,3] = PR[90,3] + 19.370;
   1:L PR[91] R[100]mm/sec CNT100;
   1:  PR[91,1] = PR[90,1] + -11.306;
   1:  PR[91,2] = PR[90,2] + 16.780;
   1:  PR[91,3] = PR[90,3] + 19.376;
   1:L PR[91] R[100]mm/sec CNT100;
   1:  PR[91,1] = PR[90,1] + -11.726;
   1:  PR[91,2] = PR[90,2] + 16.917;
   1:  PR[91,3] = PR[90,3] + 19.380;
   1:L PR[91] R[100]mm/sec CNT100;
   1:  PR[91,1] = PR[90,1] + -12.628;
   1:  PR[91,2] = PR[90,2] + 17.171;
   1:  PR[91,3] = PR[90,3] + 19.383;
   1:L PR[91] R[100]mm/sec CNT100;
   1:  PR[91,1] = PR[90,1] + -13.561;
   1:  PR[91,2] = PR[90,2] + 17.384;
   1:  PR[91,3] = PR[90,3] + 19.389;
   1:L PR[91] R[100]mm/sec CNT100;
   1:  PR[91,1] = PR[90,1] + -14.360;
   1:  PR[91,2] = PR[90,2] + 17.529;
   1:  PR[91,3] = PR[90,3] + 19.396;
   1:L PR[91] R[100]mm/sec CNT100;
   1:  PR[91,1] = PR[90,1] + -15.176;
   1:  PR[91,2] = PR[90,2] + 17.642;
   1:  PR[91,3] = PR[90,3] + 19.402;
   1:L PR[91] R[100]mm/sec CNT100;
   1:  PR[91,1] = PR[90,1] + -16.003;
   1:  PR[91,2] = PR[90,2] + 17.721;
   1:  PR[91,3] = PR[90,3] + 19.407;
   1:L PR[91] R[100]mm/sec CNT100;
   1:  PR[91,1] = PR[90,1] + -16.479;
   1:  PR[91,2] = PR[90,2] + 17.750;
   1:  PR[91,3] = PR[90,3] + 19.413;
   1:L PR[91] R[100]mm/sec CNT100;
   1:  PR[91,1] = PR[90,1] + -17.672;
   1:  PR[91,2] = PR[90,2] + 17.773;
   1:  PR[91,3] = PR[90,3] + 19.416;
   1:L PR[91] R[100]mm/sec CNT100;
   1:  PR[91,1] = PR[90,1] + -18.510;
   1:  PR[91,2] = PR[90,2] + 17.744;
   1:  PR[91,3] = PR[90,3] + 19.425;
   1:L PR[91] R[100]mm/sec CNT100;
   1:  PR[91,1] = PR[90,1] + -19.413;
   1:  PR[91,2] = PR[90,2] + 17.673;
   1:  PR[91,3] = PR[90,3] + 19.431;
   1:L PR[91] R[100]mm/sec CNT100;
   1:  PR[91,1] = PR[90,1] + -20.322;
   1:  PR[91,2] = PR[90,2] + 17.556;
   1:  PR[91,3] = PR[90,3] + 19.437;
   1:L PR[91] R[100]mm/sec CNT100;
   1:  PR[91,1] = PR[90,1] + -21.220;
   1:  PR[91,2] = PR[90,2] + 17.398;
   1:  PR[91,3] = PR[90,3] + 19.443;
   1:L PR[91] R[100]mm/sec CNT100;
   1:  PR[91,1] = PR[90,1] + -22.107;
   1:  PR[91,2] = PR[90,2] + 17.197;
   1:  PR[91,3] = PR[90,3] + 19.450;
   1:L PR[91] R[100]mm/sec CNT100;
   1:  PR[91,1] = PR[90,1] + -22.978;
   1:  PR[91,2] = PR[90,2] + 16.955;
   1:  PR[91,3] = PR[90,3] + 19.456;
   1:L PR[91] R[100]mm/sec CNT100;
   1:  PR[91,1] = PR[90,1] + -23.834;
   1:  PR[91,2] = PR[90,2] + 16.672;
   1:  PR[91,3] = PR[90,3] + 19.462;
   1:L PR[91] R[100]mm/sec CNT100;
   1:  PR[91,1] = PR[90,1] + -24.669;
   1:  PR[91,2] = PR[90,2] + 16.350;
   1:  PR[91,3] = PR[90,3] + 19.468;
   1:L PR[91] R[100]mm/sec CNT100;
   1:  PR[91,1] = PR[90,1] + -25.481;
   1:  PR[91,2] = PR[90,2] + 15.991;
   1:  PR[91,3] = PR[90,3] + 19.475;
   1:L PR[91] R[100]mm/sec CNT100;
   1:  PR[91,1] = PR[90,1] + -26.272;
   1:  PR[91,2] = PR[90,2] + 15.595;
   1:  PR[91,3] = PR[90,3] + 19.481;
   1:L PR[91] R[100]mm/sec CNT100;
   1:  PR[91,1] = PR[90,1] + -26.766;
   1:  PR[91,2] = PR[90,2] + 15.319;
   1:  PR[91,3] = PR[90,3] + 19.487;
   1:L PR[91] R[100]mm/sec CNT100;
   1:  PR[91,1] = PR[90,1] + -27.039;
   1:  PR[91,2] = PR[90,2] + 15.164;
   1:  PR[91,3] = PR[90,3] + 19.491;
   1:L PR[91] R[100]mm/sec CNT100;
   1:  PR[91,1] = PR[90,1] + -27.782;
   1:  PR[91,2] = PR[90,2] + 14.698;
   1:  PR[91,3] = PR[90,3] + 19.493;
   1:L PR[91] R[100]mm/sec CNT100;
   1:  PR[91,1] = PR[90,1] + -28.499;
   1:  PR[91,2] = PR[90,2] + 14.200;
   1:  PR[91,3] = PR[90,3] + 19.499;
   1:L PR[91] R[100]mm/sec CNT100;
   1:  PR[91,1] = PR[90,1] + -29.187;
   1:  PR[91,2] = PR[90,2] + 13.670;
   1:  PR[91,3] = PR[90,3] + 19.505;
   1:L PR[91] R[100]mm/sec CNT100;
   1:  PR[91,1] = PR[90,1] + -29.846;
   1:  PR[91,2] = PR[90,2] + 13.110;
   1:  PR[91,3] = PR[90,3] + 19.511;
   1:L PR[91] R[100]mm/sec CNT100;
   1:  PR[91,1] = PR[90,1] + -30.475;
   1:  PR[91,2] = PR[90,2] + 12.520;
   1:  PR[91,3] = PR[90,3] + 19.517;
   1:L PR[91] R[100]mm/sec CNT100;
   1:  PR[91,1] = PR[90,1] + -31.081;
   1:  PR[91,2] = PR[90,2] + 11.891;
   1:  PR[91,3] = PR[90,3] + 19.523;
   1:L PR[91] R[100]mm/sec CNT100;
   1:  PR[91,1] = PR[90,1] + -31.625;
   1:  PR[91,2] = PR[90,2] + 11.267;
   1:  PR[91,3] = PR[90,3] + 19.529;
   1:L PR[91] R[100]mm/sec CNT100;
   1:  PR[91,1] = PR[90,1] + -32.143;
   1:  PR[91,2] = PR[90,2] + 10.609;
   1:  PR[91,3] = PR[90,3] + 19.535;
   1:L PR[91] R[100]mm/sec CNT100;
   1:  PR[91,1] = PR[90,1] + -32.728;
   1:  PR[91,2] = PR[90,2] + 9.774;
   1:  PR[91,3] = PR[90,3] + 19.541;
   1:L PR[91] R[100]mm/sec CNT100;
   1:  PR[91,1] = PR[90,1] + -33.087;
   1:  PR[91,2] = PR[90,2] + 9.209;
   1:  PR[91,3] = PR[90,3] + 19.548;
   1:L PR[91] R[100]mm/sec CNT100;
   1:  PR[91,1] = PR[90,1] + -33.508;
   1:  PR[91,2] = PR[90,2] + 8.476;
   1:  PR[91,3] = PR[90,3] + 19.553;
   1:L PR[91] R[100]mm/sec CNT100;
   1:  PR[91,1] = PR[90,1] + -33.892;
   1:  PR[91,2] = PR[90,2] + 7.725;
   1:  PR[91,3] = PR[90,3] + 19.559;
   1:L PR[91] R[100]mm/sec CNT100;
   1:  PR[91,1] = PR[90,1] + -34.239;
   1:  PR[91,2] = PR[90,2] + 6.960;
   1:  PR[91,3] = PR[90,3] + 19.564;
   1:L PR[91] R[100]mm/sec CNT100;
   1:  PR[91,1] = PR[90,1] + -34.548;
   1:  PR[91,2] = PR[90,2] + 6.185;
   1:  PR[91,3] = PR[90,3] + 19.570;
   1:L PR[91] R[100]mm/sec CNT100;
   1:  PR[91,1] = PR[90,1] + -34.817;
   1:  PR[91,2] = PR[90,2] + 5.402;
   1:  PR[91,3] = PR[90,3] + 19.576;
   1:L PR[91] R[100]mm/sec CNT100;
   1:  PR[91,1] = PR[90,1] + -35.046;
   1:  PR[91,2] = PR[90,2] + 4.611;
   1:  PR[91,3] = PR[90,3] + 19.582;
   1:L PR[91] R[100]mm/sec CNT100;
   1:  PR[91,1] = PR[90,1] + -35.234;
   1:  PR[91,2] = PR[90,2] + 3.811;
   1:  PR[91,3] = PR[90,3] + 19.587;
   1:L PR[91] R[100]mm/sec CNT100;
   1:  PR[91,1] = PR[90,1] + -35.380;
   1:  PR[91,2] = PR[90,2] + 2.998;
   1:  PR[91,3] = PR[90,3] + 19.593;
   1:L PR[91] R[100]mm/sec CNT100;
   1:  PR[91,1] = PR[90,1] + -35.486;
   1:  PR[91,2] = PR[90,2] + 2.166;
   1:  PR[91,3] = PR[90,3] + 19.599;
   1:L PR[91] R[100]mm/sec CNT100;
   1:  PR[91,1] = PR[90,1] + -35.549;
   1:  PR[91,2] = PR[90,2] + 1.310;
   1:  PR[91,3] = PR[90,3] + 19.605;
   1:L PR[91] R[100]mm/sec CNT100;
   1:  PR[91,1] = PR[90,1] + -35.570;
   1:  PR[91,2] = PR[90,2] + 0.428;
   1:  PR[91,3] = PR[90,3] + 19.611;
   1:L PR[91] R[100]mm/sec CNT100;
   1:  PR[91,1] = PR[90,1] + -35.549;
   1:  PR[91,2] = PR[90,2] + -0.455;
   1:  PR[91,3] = PR[90,3] + 19.617;
   1:L PR[91] R[100]mm/sec CNT100;
   1:  PR[91,1] = PR[90,1] + -35.486;
   1:  PR[91,2] = PR[90,2] + -1.311;
   1:  PR[91,3] = PR[90,3] + 19.623;
   1:L PR[91] R[100]mm/sec CNT100;
   1:  PR[91,1] = PR[90,1] + -35.380;
   1:  PR[91,2] = PR[90,2] + -2.143;
   1:  PR[91,3] = PR[90,3] + 19.629;
   1:L PR[91] R[100]mm/sec CNT100;
   1:  PR[91,1] = PR[90,1] + -35.234;
   1:  PR[91,2] = PR[90,2] + -2.956;
   1:  PR[91,3] = PR[90,3] + 19.635;
   1:L PR[91] R[100]mm/sec CNT100;
   1:  PR[91,1] = PR[90,1] + -35.046;
   1:  PR[91,2] = PR[90,2] + -3.756;
   1:  PR[91,3] = PR[90,3] + 19.641;
   1:L PR[91] R[100]mm/sec CNT100;
   1:  PR[91,1] = PR[90,1] + -34.817;
   1:  PR[91,2] = PR[90,2] + -4.547;
   1:  PR[91,3] = PR[90,3] + 19.646;
   1:L PR[91] R[100]mm/sec CNT100;
   1:  PR[91,1] = PR[90,1] + -34.548;
   1:  PR[91,2] = PR[90,2] + -5.330;
   1:  PR[91,3] = PR[90,3] + 19.652;
   1:L PR[91] R[100]mm/sec CNT100;
   1:  PR[91,1] = PR[90,1] + -34.239;
   1:  PR[91,2] = PR[90,2] + -6.104;
   1:  PR[91,3] = PR[90,3] + 19.658;
   1:L PR[91] R[100]mm/sec CNT100;
   1:  PR[91,1] = PR[90,1] + -33.892;
   1:  PR[91,2] = PR[90,2] + -6.870;
   1:  PR[91,3] = PR[90,3] + 19.664;
   1:L PR[91] R[100]mm/sec CNT100;
   1:  PR[91,1] = PR[90,1] + -33.630;
   1:  PR[91,2] = PR[90,2] + -7.384;
   1:  PR[91,3] = PR[90,3] + 19.669;
   1:L PR[91] R[100]mm/sec CNT100;
   1:  PR[91,1] = PR[90,1] + -33.508;
   1:  PR[91,2] = PR[90,2] + -7.620;
   1:  PR[91,3] = PR[90,3] + 19.673;
   1:L PR[91] R[100]mm/sec CNT100;
   1:  PR[91,1] = PR[90,1] + -33.087;
   1:  PR[91,2] = PR[90,2] + -8.354;
   1:  PR[91,3] = PR[90,3] + 19.675;
   1:L PR[91] R[100]mm/sec CNT100;
   1:  PR[91,1] = PR[90,1] + -32.728;
   1:  PR[91,2] = PR[90,2] + -8.918;
   1:  PR[91,3] = PR[90,3] + 19.681;
   1:L PR[91] R[100]mm/sec CNT100;
   1:  PR[91,1] = PR[90,1] + -32.143;
   1:  PR[91,2] = PR[90,2] + -9.754;
   1:  PR[91,3] = PR[90,3] + 19.686;
   1:L PR[91] R[100]mm/sec CNT100;
   1:  PR[91,1] = PR[90,1] + -31.625;
   1:  PR[91,2] = PR[90,2] + -10.412;
   1:  PR[91,3] = PR[90,3] + 19.693;
   1:L PR[91] R[100]mm/sec CNT100;
   1:  PR[91,1] = PR[90,1] + -31.071;
   1:  PR[91,2] = PR[90,2] + -11.047;
   1:  PR[91,3] = PR[90,3] + 19.699;
   1:L PR[91] R[100]mm/sec CNT100;
   1:  PR[91,1] = PR[90,1] + -30.475;
   1:  PR[91,2] = PR[90,2] + -11.665;
   1:  PR[91,3] = PR[90,3] + 19.705;
   1:L PR[91] R[100]mm/sec CNT100;
   1:  PR[91,1] = PR[90,1] + -29.846;
   1:  PR[91,2] = PR[90,2] + -12.254;
   1:  PR[91,3] = PR[90,3] + 19.710;
   1:L PR[91] R[100]mm/sec CNT100;
   1:  PR[91,1] = PR[90,1] + -29.187;
   1:  PR[91,2] = PR[90,2] + -12.815;
   1:  PR[91,3] = PR[90,3] + 19.716;
   1:L PR[91] R[100]mm/sec CNT100;
   1:  PR[91,1] = PR[90,1] + -28.499;
   1:  PR[91,2] = PR[90,2] + -13.345;
   1:  PR[91,3] = PR[90,3] + 19.722;
   1:L PR[91] R[100]mm/sec CNT100;
   1:  PR[91,1] = PR[90,1] + -27.782;
   1:  PR[91,2] = PR[90,2] + -13.843;
   1:  PR[91,3] = PR[90,3] + 19.729;
   1:L PR[91] R[100]mm/sec CNT100;
   1:  PR[91,1] = PR[90,1] + -27.039;
   1:  PR[91,2] = PR[90,2] + -14.309;
   1:  PR[91,3] = PR[90,3] + 19.735;
   1:L PR[91] R[100]mm/sec CNT100;
   1:  PR[91,1] = PR[90,1] + -26.766;
   1:  PR[91,2] = PR[90,2] + -14.463;
   1:  PR[91,3] = PR[90,3] + 19.741;
   1:L PR[91] R[100]mm/sec CNT100;
   1:  PR[91,1] = PR[90,1] + -26.272;
   1:  PR[91,2] = PR[90,2] + -14.740;
   1:  PR[91,3] = PR[90,3] + 19.743;
   1:L PR[91] R[100]mm/sec CNT100;
   1:  PR[91,1] = PR[90,1] + -25.481;
   1:  PR[91,2] = PR[90,2] + -15.136;
   1:  PR[91,3] = PR[90,3] + 19.747;
   1:L PR[91] R[100]mm/sec CNT100;
   1:  PR[91,1] = PR[90,1] + -24.669;
   1:  PR[91,2] = PR[90,2] + -15.495;
   1:  PR[91,3] = PR[90,3] + 19.753;
   1:L PR[91] R[100]mm/sec CNT100;
   1:  PR[91,1] = PR[90,1] + -23.834;
   1:  PR[91,2] = PR[90,2] + -15.817;
   1:  PR[91,3] = PR[90,3] + 19.759;
   1:L PR[91] R[100]mm/sec CNT100;
   1:  PR[91,1] = PR[90,1] + -22.978;
   1:  PR[91,2] = PR[90,2] + -16.100;
   1:  PR[91,3] = PR[90,3] + 19.765;
   1:L PR[91] R[100]mm/sec CNT100;
   1:  PR[91,1] = PR[90,1] + -22.107;
   1:  PR[91,2] = PR[90,2] + -16.342;
   1:  PR[91,3] = PR[90,3] + 19.772;
   1:L PR[91] R[100]mm/sec CNT100;
   1:  PR[91,1] = PR[90,1] + -21.220;
   1:  PR[91,2] = PR[90,2] + -16.543;
   1:  PR[91,3] = PR[90,3] + 19.778;
   1:L PR[91] R[100]mm/sec CNT100;
   1:  PR[91,1] = PR[90,1] + -20.322;
   1:  PR[91,2] = PR[90,2] + -16.701;
   1:  PR[91,3] = PR[90,3] + 19.784;
   1:L PR[91] R[100]mm/sec CNT100;
   1:  PR[91,1] = PR[90,1] + -19.413;
   1:  PR[91,2] = PR[90,2] + -16.817;
   1:  PR[91,3] = PR[90,3] + 19.791;
   1:L PR[91] R[100]mm/sec CNT100;
   1:  PR[91,1] = PR[90,1] + -18.481;
   1:  PR[91,2] = PR[90,2] + -16.891;
   1:  PR[91,3] = PR[90,3] + 19.797;
   1:L PR[91] R[100]mm/sec CNT100;
   1:  PR[91,1] = PR[90,1] + -17.672;
   1:  PR[91,2] = PR[90,2] + -16.918;
   1:  PR[91,3] = PR[90,3] + 19.803;
   1:L PR[91] R[100]mm/sec CNT100;
   1:  PR[91,1] = PR[90,1] + -16.479;
   1:  PR[91,2] = PR[90,2] + -16.895;
   1:  PR[91,3] = PR[90,3] + 19.809;
   1:L PR[91] R[100]mm/sec CNT100;
   1:  PR[91,1] = PR[90,1] + -16.003;
   1:  PR[91,2] = PR[90,2] + -16.866;
   1:  PR[91,3] = PR[90,3] + 19.817;
   1:L PR[91] R[100]mm/sec CNT100;
   1:  PR[91,1] = PR[90,1] + -15.176;
   1:  PR[91,2] = PR[90,2] + -16.787;
   1:  PR[91,3] = PR[90,3] + 19.821;
   1:L PR[91] R[100]mm/sec CNT100;
   1:  PR[91,1] = PR[90,1] + -14.360;
   1:  PR[91,2] = PR[90,2] + -16.674;
   1:  PR[91,3] = PR[90,3] + 19.826;
   1:L PR[91] R[100]mm/sec CNT100;
   1:  PR[91,1] = PR[90,1] + -13.539;
   1:  PR[91,2] = PR[90,2] + -16.525;
   1:  PR[91,3] = PR[90,3] + 19.832;
   1:L PR[91] R[100]mm/sec CNT100;
   1:  PR[91,1] = PR[90,1] + -12.628;
   1:  PR[91,2] = PR[90,2] + -16.316;
   1:  PR[91,3] = PR[90,3] + 19.838;
   1:L PR[91] R[100]mm/sec CNT100;
   1:  PR[91,1] = PR[90,1] + -11.726;
   1:  PR[91,2] = PR[90,2] + -16.062;
   1:  PR[91,3] = PR[90,3] + 19.844;
   1:L PR[91] R[100]mm/sec CNT100;
   1:  PR[91,1] = PR[90,1] + -11.306;
   1:  PR[91,2] = PR[90,2] + -15.925;
   1:  PR[91,3] = PR[90,3] + 19.851;
   1:L PR[91] R[100]mm/sec CNT100;
   1:  PR[91,1] = PR[90,1] + -10.841;
   1:  PR[91,2] = PR[90,2] + -15.766;
   1:  PR[91,3] = PR[90,3] + 19.854;
   1:L PR[91] R[100]mm/sec CNT100;
   1:  PR[91,1] = PR[90,1] + -9.965;
   1:  PR[91,2] = PR[90,2] + -15.424;
   1:  PR[91,3] = PR[90,3] + 19.857;
   1:L PR[91] R[100]mm/sec CNT100;
   1:  PR[91,1] = PR[90,1] + -9.096;
   1:  PR[91,2] = PR[90,2] + -15.035;
   1:  PR[91,3] = PR[90,3] + 19.864;
   1:L PR[91] R[100]mm/sec CNT100;
   1:  PR[91,1] = PR[90,1] + -8.279;
   1:  PR[91,2] = PR[90,2] + -14.622;
   1:  PR[91,3] = PR[90,3] + 19.871;
   1:L PR[91] R[100]mm/sec CNT100;
   1:  PR[91,1] = PR[90,1] + -7.577;
   1:  PR[91,2] = PR[90,2] + -14.226;
   1:  PR[91,3] = PR[90,3] + 19.877;
   1:L PR[91] R[100]mm/sec CNT100;
   1:  PR[91,1] = PR[90,1] + -6.624;
   1:  PR[91,2] = PR[90,2] + -13.622;
   1:  PR[91,3] = PR[90,3] + 19.883;
   1:L PR[91] R[100]mm/sec CNT100;
   1:  PR[91,1] = PR[90,1] + -6.044;
   1:  PR[91,2] = PR[90,2] + -13.213;
   1:  PR[91,3] = PR[90,3] + 19.890;
   1:L PR[91] R[100]mm/sec CNT100;
   1:  PR[91,1] = PR[90,1] + -5.542;
   1:  PR[91,2] = PR[90,2] + -12.831;
   1:  PR[91,3] = PR[90,3] + 19.895;
   1:L PR[91] R[100]mm/sec CNT100;
   1:  PR[91,1] = PR[90,1] + -5.052;
   1:  PR[91,2] = PR[90,2] + -12.431;
   1:  PR[91,3] = PR[90,3] + 19.900;
   1:L PR[91] R[100]mm/sec CNT100;
   1:  PR[91,1] = PR[90,1] + -4.606;
   1:  PR[91,2] = PR[90,2] + -12.042;
   1:  PR[91,3] = PR[90,3] + 19.904;
   1:L PR[91] R[100]mm/sec CNT100;
   1:  PR[91,1] = PR[90,1] + -4.134;
   1:  PR[91,2] = PR[90,2] + -11.600;
   1:  PR[91,3] = PR[90,3] + 19.908;
   1:L PR[91] R[100]mm/sec CNT100;
   1:  PR[91,1] = PR[90,1] + -3.299;
   1:  PR[91,2] = PR[90,2] + -10.730;
   1:  PR[91,3] = PR[90,3] + 19.913;
   1:L PR[91] R[100]mm/sec CNT100;
   1:  PR[91,1] = PR[90,1] + -2.933;
   1:  PR[91,2] = PR[90,2] + -10.305;
   1:  PR[91,3] = PR[90,3] + 19.921;
   1:L PR[91] R[100]mm/sec CNT100;
   1:  PR[91,1] = PR[90,1] + -2.436;
   1:  PR[91,2] = PR[90,2] + -9.678;
   1:  PR[91,3] = PR[90,3] + 19.925;
   1:L PR[91] R[100]mm/sec CNT100;
   1:  PR[91,1] = PR[90,1] + -2.119;
   1:  PR[91,2] = PR[90,2] + -9.308;
   1:  PR[91,3] = PR[90,3] + 19.931;
   1:L PR[91] R[100]mm/sec CNT100;
   1:  PR[91,1] = PR[90,1] + -1.727;
   1:  PR[91,2] = PR[90,2] + -8.984;
   1:  PR[91,3] = PR[90,3] + 19.934;
   1:L PR[91] R[100]mm/sec CNT100;
   1:  PR[91,1] = PR[90,1] + -1.293;
   1:  PR[91,2] = PR[90,2] + -8.732;
   1:  PR[91,3] = PR[90,3] + 19.937;
   1:L PR[91] R[100]mm/sec CNT100;
   1:  PR[91,1] = PR[90,1] + -0.824;
   1:  PR[91,2] = PR[90,2] + -8.560;
   1:  PR[91,3] = PR[90,3] + 19.941;
   1:L PR[91] R[100]mm/sec CNT100;
   1:  PR[91,1] = PR[90,1] + -0.336;
   1:  PR[91,2] = PR[90,2] + -8.475;
   1:  PR[91,3] = PR[90,3] + 19.944;
   1:L PR[91] R[100]mm/sec CNT100;
   1:  PR[91,1] = PR[90,1] + -0.027;
   1:  PR[91,2] = PR[90,2] + -8.473;
   1:  PR[91,3] = PR[90,3] + 19.948;
   1:L PR[91] R[100]mm/sec CNT100;
   1:  PR[91] = PR[90];
   1:  PR[91,1] = PR[90,1] + 0.301;
   1:  PR[91,2] = PR[90,2] + -9.335;
   1:  PR[91,3] = PR[90,3] + 21.280;
   1:L PR[91] R[100]mm/sec CNT100;
   1:  PR[91,1] = PR[90,1] + 0.793;
   1:  PR[91,2] = PR[90,2] + -9.456;
   1:  PR[91,3] = PR[90,3] + 19.954;
   1:L PR[91] R[100]mm/sec CNT100;
   1:  PR[91,1] = PR[90,1] + 1.261;
   1:  PR[91,2] = PR[90,2] + -9.666;
   1:  PR[91,3] = PR[90,3] + 19.957;
   1:L PR[91] R[100]mm/sec CNT100;
   1:  PR[91,1] = PR[90,1] + 1.691;
   1:  PR[91,2] = PR[90,2] + -9.957;
   1:  PR[91,3] = PR[90,3] + 19.961;
   1:L PR[91] R[100]mm/sec CNT100;
   1:  PR[91,1] = PR[90,1] + 2.059;
   1:  PR[91,2] = PR[90,2] + -10.310;
   1:  PR[91,3] = PR[90,3] + 19.964;
   1:L PR[91] R[100]mm/sec CNT100;
   1:  PR[91,1] = PR[90,1] + 2.528;
   1:  PR[91,2] = PR[90,2] + -10.862;
   1:  PR[91,3] = PR[90,3] + 19.968;
   1:L PR[91] R[100]mm/sec CNT100;
   1:  PR[91,1] = PR[90,1] + 3.083;
   1:  PR[91,2] = PR[90,2] + -11.450;
   1:  PR[91,3] = PR[90,3] + 19.973;
   1:L PR[91] R[100]mm/sec CNT100;
   1:  PR[91,1] = PR[90,1] + 3.853;
   1:  PR[91,2] = PR[90,2] + -12.187;
   1:  PR[91,3] = PR[90,3] + 19.979;
   1:L PR[91] R[100]mm/sec CNT100;
   1:  PR[91,1] = PR[90,1] + 4.697;
   1:  PR[91,2] = PR[90,2] + -12.898;
   1:  PR[91,3] = PR[90,3] + 19.986;
   1:L PR[91] R[100]mm/sec CNT100;
   1:  PR[91,1] = PR[90,1] + 5.304;
   1:  PR[91,2] = PR[90,2] + -13.358;
   1:  PR[91,3] = PR[90,3] + 19.994;
   1:L PR[91] R[100]mm/sec CNT100;
   1:  PR[91,1] = PR[90,1] + 5.906;
   1:  PR[91,2] = PR[90,2] + -13.774;
   1:  PR[91,3] = PR[90,3] + 19.999;
   1:L PR[91] R[100]mm/sec CNT100;
   1:  PR[91,1] = PR[90,1] + 6.879;
   1:  PR[91,2] = PR[90,2] + -14.379;
   1:  PR[91,3] = PR[90,3] + 20.005;
   1:L PR[91] R[100]mm/sec CNT100;
   1:  PR[91,1] = PR[90,1] + 7.941;
   1:  PR[91,2] = PR[90,2] + -14.950;
   1:  PR[91,3] = PR[90,3] + 20.013;
   1:L PR[91] R[100]mm/sec CNT100;
   1:  PR[91,1] = PR[90,1] + 8.559;
   1:  PR[91,2] = PR[90,2] + -15.244;
   1:  PR[91,3] = PR[90,3] + 20.021;
   1:L PR[91] R[100]mm/sec CNT100;
   1:  PR[91,1] = PR[90,1] + 9.095;
   1:  PR[91,2] = PR[90,2] + -15.477;
   1:  PR[91,3] = PR[90,3] + 20.026;
   1:L PR[91] R[100]mm/sec CNT100;
   1:  PR[91,1] = PR[90,1] + 9.725;
   1:  PR[91,2] = PR[90,2] + -15.727;
   1:  PR[91,3] = PR[90,3] + 20.030;
   1:L PR[91] R[100]mm/sec CNT100;
   1:  PR[91,1] = PR[90,1] + 10.302;
   1:  PR[91,2] = PR[90,2] + -15.935;
   1:  PR[91,3] = PR[90,3] + 20.035;
   1:L PR[91] R[100]mm/sec CNT100;
   1:  PR[91,1] = PR[90,1] + 10.923;
   1:  PR[91,2] = PR[90,2] + -16.137;
   1:  PR[91,3] = PR[90,3] + 20.039;
   1:L PR[91] R[100]mm/sec CNT100;
   1:  PR[91,1] = PR[90,1] + 11.965;
   1:  PR[91,2] = PR[90,2] + -16.425;
   1:  PR[91,3] = PR[90,3] + 20.044;
   1:L PR[91] R[100]mm/sec CNT100;
   1:  PR[91,1] = PR[90,1] + 12.689;
   1:  PR[91,2] = PR[90,2] + -16.591;
   1:  PR[91,3] = PR[90,3] + 20.051;
   1:L PR[91] R[100]mm/sec CNT100;
   1:  PR[91,1] = PR[90,1] + 13.512;
   1:  PR[91,2] = PR[90,2] + -16.744;
   1:  PR[91,3] = PR[90,3] + 20.057;
   1:L PR[91] R[100]mm/sec CNT100;
   1:  PR[91,1] = PR[90,1] + 14.436;
   1:  PR[91,2] = PR[90,2] + -16.874;
   1:  PR[91,3] = PR[90,3] + 20.062;
   1:L PR[91] R[100]mm/sec CNT100;
   1:  PR[91,1] = PR[90,1] + 15.372;
   1:  PR[91,2] = PR[90,2] + -16.960;
   1:  PR[91,3] = PR[90,3] + 20.069;
   1:L PR[91] R[100]mm/sec CNT100;
   1:  PR[91,1] = PR[90,1] + 16.309;
   1:  PR[91,2] = PR[90,2] + -17.001;
   1:  PR[91,3] = PR[90,3] + 20.076;
   1:L PR[91] R[100]mm/sec CNT100;
   1:  PR[91,1] = PR[90,1] + 16.710;
   1:  PR[91,2] = PR[90,2] + -17.002;
   1:  PR[91,3] = PR[90,3] + 20.082;
   1:L PR[91] R[100]mm/sec CNT100;
   1:  PR[91,1] = PR[90,1] + 17.239;
   1:  PR[91,2] = PR[90,2] + -16.998;
   1:  PR[91,3] = PR[90,3] + 20.085;
   1:L PR[91] R[100]mm/sec CNT100;
   1:  PR[91,1] = PR[90,1] + 18.169;
   1:  PR[91,2] = PR[90,2] + -16.950;
   1:  PR[91,3] = PR[90,3] + 20.089;
   1:L PR[91] R[100]mm/sec CNT100;
   1:  PR[91,1] = PR[90,1] + 19.065;
   1:  PR[91,2] = PR[90,2] + -16.862;
   1:  PR[91,3] = PR[90,3] + 20.095;
   1:L PR[91] R[100]mm/sec CNT100;
   1:  PR[91,1] = PR[90,1] + 19.893;
   1:  PR[91,2] = PR[90,2] + -16.743;
   1:  PR[91,3] = PR[90,3] + 20.102;
   1:L PR[91] R[100]mm/sec CNT100;
   1:  PR[91,1] = PR[90,1] + 20.719;
   1:  PR[91,2] = PR[90,2] + -16.588;
   1:  PR[91,3] = PR[90,3] + 20.108;
   1:L PR[91] R[100]mm/sec CNT100;
   1:  PR[91,1] = PR[90,1] + 21.541;
   1:  PR[91,2] = PR[90,2] + -16.395;
   1:  PR[91,3] = PR[90,3] + 20.114;
   1:L PR[91] R[100]mm/sec CNT100;
   1:  PR[91,1] = PR[90,1] + 22.357;
   1:  PR[91,2] = PR[90,2] + -16.166;
   1:  PR[91,3] = PR[90,3] + 20.119;
   1:L PR[91] R[100]mm/sec CNT100;
   1:  PR[91,1] = PR[90,1] + 23.165;
   1:  PR[91,2] = PR[90,2] + -15.900;
   1:  PR[91,3] = PR[90,3] + 20.125;
   1:L PR[91] R[100]mm/sec CNT100;
   1:  PR[91,1] = PR[90,1] + 23.963;
   1:  PR[91,2] = PR[90,2] + -15.598;
   1:  PR[91,3] = PR[90,3] + 20.131;
   1:L PR[91] R[100]mm/sec CNT100;
   1:  PR[91,1] = PR[90,1] + 24.775;
   1:  PR[91,2] = PR[90,2] + -15.247;
   1:  PR[91,3] = PR[90,3] + 20.137;
   1:L PR[91] R[100]mm/sec CNT100;
   1:  PR[91,1] = PR[90,1] + 25.582;
   1:  PR[91,2] = PR[90,2] + -14.851;
   1:  PR[91,3] = PR[90,3] + 20.144;
   1:L PR[91] R[100]mm/sec CNT100;
   1:  PR[91,1] = PR[90,1] + 26.365;
   1:  PR[91,2] = PR[90,2] + -14.419;
   1:  PR[91,3] = PR[90,3] + 20.150;
   1:L PR[91] R[100]mm/sec CNT100;
   1:  PR[91,1] = PR[90,1] + 27.123;
   1:  PR[91,2] = PR[90,2] + -13.951;
   1:  PR[91,3] = PR[90,3] + 20.156;
   1:L PR[91] R[100]mm/sec CNT100;
   1:  PR[91,1] = PR[90,1] + 27.853;
   1:  PR[91,2] = PR[90,2] + -13.451;
   1:  PR[91,3] = PR[90,3] + 20.163;
   1:L PR[91] R[100]mm/sec CNT100;
   1:  PR[91,1] = PR[90,1] + 28.555;
   1:  PR[91,2] = PR[90,2] + -12.918;
   1:  PR[91,3] = PR[90,3] + 20.169;
   1:L PR[91] R[100]mm/sec CNT100;
   1:  PR[91,1] = PR[90,1] + 29.227;
   1:  PR[91,2] = PR[90,2] + -12.353;
   1:  PR[91,3] = PR[90,3] + 20.175;
   1:L PR[91] R[100]mm/sec CNT100;
   1:  PR[91,1] = PR[90,1] + 29.867;
   1:  PR[91,2] = PR[90,2] + -11.758;
   1:  PR[91,3] = PR[90,3] + 20.181;
   1:L PR[91] R[100]mm/sec CNT100;
   1:  PR[91,1] = PR[90,1] + 30.477;
   1:  PR[91,2] = PR[90,2] + -11.131;
   1:  PR[91,3] = PR[90,3] + 20.187;
   1:L PR[91] R[100]mm/sec CNT100;
   1:  PR[91,1] = PR[90,1] + 31.046;
   1:  PR[91,2] = PR[90,2] + -10.482;
   1:  PR[91,3] = PR[90,3] + 20.193;
   1:L PR[91] R[100]mm/sec CNT100;
   1:  PR[91,1] = PR[90,1] + 31.582;
   1:  PR[91,2] = PR[90,2] + -9.804;
   1:  PR[91,3] = PR[90,3] + 20.200;
   1:L PR[91] R[100]mm/sec CNT100;
   1:  PR[91,1] = PR[90,1] + 32.084;
   1:  PR[91,2] = PR[90,2] + -9.101;
   1:  PR[91,3] = PR[90,3] + 20.206;
   1:L PR[91] R[100]mm/sec CNT100;
   1:  PR[91,1] = PR[90,1] + 32.549;
   1:  PR[91,2] = PR[90,2] + -8.377;
   1:  PR[91,3] = PR[90,3] + 20.212;
   1:L PR[91] R[100]mm/sec CNT100;
   1:  PR[91,1] = PR[90,1] + 32.977;
   1:  PR[91,2] = PR[90,2] + -7.635;
   1:  PR[91,3] = PR[90,3] + 20.218;
   1:L PR[91] R[100]mm/sec CNT100;
   1:  PR[91,1] = PR[90,1] + 33.367;
   1:  PR[91,2] = PR[90,2] + -6.879;
   1:  PR[91,3] = PR[90,3] + 20.224;
   1:L PR[91] R[100]mm/sec CNT100;
   1:  PR[91,1] = PR[90,1] + 33.718;
   1:  PR[91,2] = PR[90,2] + -6.113;
   1:  PR[91,3] = PR[90,3] + 20.230;
   1:L PR[91] R[100]mm/sec CNT100;
   1:  PR[91,1] = PR[90,1] + 34.029;
   1:  PR[91,2] = PR[90,2] + -5.339;
   1:  PR[91,3] = PR[90,3] + 20.236;
   1:L PR[91] R[100]mm/sec CNT100;
   1:  PR[91,1] = PR[90,1] + 34.299;
   1:  PR[91,2] = PR[90,2] + -4.559;
   1:  PR[91,3] = PR[90,3] + 20.242;
   1:L PR[91] R[100]mm/sec CNT100;
   1:  PR[91,1] = PR[90,1] + 34.528;
   1:  PR[91,2] = PR[90,2] + -3.770;
   1:  PR[91,3] = PR[90,3] + 20.247;
   1:L PR[91] R[100]mm/sec CNT100;
   1:  PR[91,1] = PR[90,1] + 34.716;
   1:  PR[91,2] = PR[90,2] + -2.969;
   1:  PR[91,3] = PR[90,3] + 20.253;
   1:L PR[91] R[100]mm/sec CNT100;
   1:  PR[91,1] = PR[90,1] + 34.863;
   1:  PR[91,2] = PR[90,2] + -2.154;
   1:  PR[91,3] = PR[90,3] + 20.259;
   1:L PR[91] R[100]mm/sec CNT100;
   1:  PR[91,1] = PR[90,1] + 34.968;
   1:  PR[91,2] = PR[90,2] + -1.318;
   1:  PR[91,3] = PR[90,3] + 20.265;
   1:L PR[91] R[100]mm/sec CNT100;
   1:  PR[91,1] = PR[90,1] + 35.031;
   1:  PR[91,2] = PR[90,2] + -0.458;
   1:  PR[91,3] = PR[90,3] + 20.271;
   1:L PR[91] R[100]mm/sec CNT100;
   1:  PR[91,1] = PR[90,1] + 35.055;
   1:  PR[91,2] = PR[90,2] + 0.428;
   1:  PR[91,3] = PR[90,3] + 20.277;
   1:L PR[91] R[100]mm/sec CNT100;
   1:  PR[91,1] = PR[90,1] + 35.031;
   1:  PR[91,2] = PR[90,2] + 1.313;
   1:  PR[91,3] = PR[90,3] + 20.283;
   1:L PR[91] R[100]mm/sec CNT100;
   1:  PR[91,1] = PR[90,1] + 34.968;
   1:  PR[91,2] = PR[90,2] + 2.173;
   1:  PR[91,3] = PR[90,3] + 20.289;
   1:L PR[91] R[100]mm/sec CNT100;
   1:  PR[91,1] = PR[90,1] + 34.863;
   1:  PR[91,2] = PR[90,2] + 3.009;
   1:  PR[91,3] = PR[90,3] + 20.295;
   1:L PR[91] R[100]mm/sec CNT100;
   1:  PR[91,1] = PR[90,1] + 34.716;
   1:  PR[91,2] = PR[90,2] + 3.825;
   1:  PR[91,3] = PR[90,3] + 20.301;
   1:L PR[91] R[100]mm/sec CNT100;
   1:  PR[91,1] = PR[90,1] + 34.528;
   1:  PR[91,2] = PR[90,2] + 4.625;
   1:  PR[91,3] = PR[90,3] + 20.307;
   1:L PR[91] R[100]mm/sec CNT100;
   1:  PR[91,1] = PR[90,1] + 34.299;
   1:  PR[91,2] = PR[90,2] + 5.414;
   1:  PR[91,3] = PR[90,3] + 20.313;
   1:L PR[91] R[100]mm/sec CNT100;
   1:  PR[91,1] = PR[90,1] + 34.029;
   1:  PR[91,2] = PR[90,2] + 6.194;
   1:  PR[91,3] = PR[90,3] + 20.319;
   1:L PR[91] R[100]mm/sec CNT100;
   1:  PR[91,1] = PR[90,1] + 33.718;
   1:  PR[91,2] = PR[90,2] + 6.968;
   1:  PR[91,3] = PR[90,3] + 20.325;
   1:L PR[91] R[100]mm/sec CNT100;
   1:  PR[91,1] = PR[90,1] + 33.367;
   1:  PR[91,2] = PR[90,2] + 7.734;
   1:  PR[91,3] = PR[90,3] + 20.330;
   1:L PR[91] R[100]mm/sec CNT100;
   1:  PR[91,1] = PR[90,1] + 32.977;
   1:  PR[91,2] = PR[90,2] + 8.490;
   1:  PR[91,3] = PR[90,3] + 20.336;
   1:L PR[91] R[100]mm/sec CNT100;
   1:  PR[91,1] = PR[90,1] + 32.549;
   1:  PR[91,2] = PR[90,2] + 9.232;
   1:  PR[91,3] = PR[90,3] + 20.342;
   1:L PR[91] R[100]mm/sec CNT100;
   1:  PR[91,1] = PR[90,1] + 32.084;
   1:  PR[91,2] = PR[90,2] + 9.956;
   1:  PR[91,3] = PR[90,3] + 20.348;
   1:L PR[91] R[100]mm/sec CNT100;
   1:  PR[91,1] = PR[90,1] + 31.582;
   1:  PR[91,2] = PR[90,2] + 10.658;
   1:  PR[91,3] = PR[90,3] + 20.354;
   1:L PR[91] R[100]mm/sec CNT100;
   1:  PR[91,1] = PR[90,1] + 31.046;
   1:  PR[91,2] = PR[90,2] + 11.337;
   1:  PR[91,3] = PR[90,3] + 20.361;
   1:L PR[91] R[100]mm/sec CNT100;
   1:  PR[91,1] = PR[90,1] + 30.474;
   1:  PR[91,2] = PR[90,2] + 11.989;
   1:  PR[91,3] = PR[90,3] + 20.367;
   1:L PR[91] R[100]mm/sec CNT100;
   1:  PR[91,1] = PR[90,1] + 29.867;
   1:  PR[91,2] = PR[90,2] + 12.613;
   1:  PR[91,3] = PR[90,3] + 20.373;
   1:L PR[91] R[100]mm/sec CNT100;
   1:  PR[91,1] = PR[90,1] + 29.227;
   1:  PR[91,2] = PR[90,2] + 13.208;
   1:  PR[91,3] = PR[90,3] + 20.379;
   1:L PR[91] R[100]mm/sec CNT100;
   1:  PR[91,1] = PR[90,1] + 28.555;
   1:  PR[91,2] = PR[90,2] + 13.773;
   1:  PR[91,3] = PR[90,3] + 20.385;
   1:L PR[91] R[100]mm/sec CNT100;
   1:  PR[91,1] = PR[90,1] + 27.852;
   1:  PR[91,2] = PR[90,2] + 14.306;
   1:  PR[91,3] = PR[90,3] + 20.391;
   1:L PR[91] R[100]mm/sec CNT100;
   1:  PR[91,1] = PR[90,1] + 27.464;
   1:  PR[91,2] = PR[90,2] + 14.574;
   1:  PR[91,3] = PR[90,3] + 20.397;
   1:L PR[91] R[100]mm/sec CNT100;
   1:  PR[91,1] = PR[90,1] + 27.124;
   1:  PR[91,2] = PR[90,2] + 14.806;
   1:  PR[91,3] = PR[90,3] + 20.401;
   1:L PR[91] R[100]mm/sec CNT100;
   1:  PR[91,1] = PR[90,1] + 26.366;
   1:  PR[91,2] = PR[90,2] + 15.274;
   1:  PR[91,3] = PR[90,3] + 20.404;
   1:L PR[91] R[100]mm/sec CNT100;
   1:  PR[91,1] = PR[90,1] + 25.582;
   1:  PR[91,2] = PR[90,2] + 15.706;
   1:  PR[91,3] = PR[90,3] + 20.410;
   1:L PR[91] R[100]mm/sec CNT100;
   1:  PR[91,1] = PR[90,1] + 24.775;
   1:  PR[91,2] = PR[90,2] + 16.102;
   1:  PR[91,3] = PR[90,3] + 20.416;
   1:L PR[91] R[100]mm/sec CNT100;
   1:  PR[91,1] = PR[90,1] + 23.963;
   1:  PR[91,2] = PR[90,2] + 16.453;
   1:  PR[91,3] = PR[90,3] + 20.422;
   1:L PR[91] R[100]mm/sec CNT100;
   1:  PR[91,1] = PR[90,1] + 23.168;
   1:  PR[91,2] = PR[90,2] + 16.755;
   1:  PR[91,3] = PR[90,3] + 20.429;
   1:L PR[91] R[100]mm/sec CNT100;
   1:  PR[91,1] = PR[90,1] + 22.034;
   1:  PR[91,2] = PR[90,2] + 17.115;
   1:  PR[91,3] = PR[90,3] + 20.435;
   1:L PR[91] R[100]mm/sec CNT100;
   1:  PR[91,1] = PR[90,1] + 21.542;
   1:  PR[91,2] = PR[90,2] + 17.250;
   1:  PR[91,3] = PR[90,3] + 20.443;
   1:L PR[91] R[100]mm/sec CNT100;
   1:  PR[91,1] = PR[90,1] + 20.719;
   1:  PR[91,2] = PR[90,2] + 17.443;
   1:  PR[91,3] = PR[90,3] + 20.447;
   1:L PR[91] R[100]mm/sec CNT100;
   1:  PR[91,1] = PR[90,1] + 19.893;
   1:  PR[91,2] = PR[90,2] + 17.599;
   1:  PR[91,3] = PR[90,3] + 20.453;
   1:L PR[91] R[100]mm/sec CNT100;
   1:  PR[91,1] = PR[90,1] + 19.065;
   1:  PR[91,2] = PR[90,2] + 17.718;
   1:  PR[91,3] = PR[90,3] + 20.459;
   1:L PR[91] R[100]mm/sec CNT100;
   1:  PR[91,1] = PR[90,1] + 18.168;
   1:  PR[91,2] = PR[90,2] + 17.805;
   1:  PR[91,3] = PR[90,3] + 20.464;
   1:L PR[91] R[100]mm/sec CNT100;
   1:  PR[91,1] = PR[90,1] + 17.496;
   1:  PR[91,2] = PR[90,2] + 17.841;
   1:  PR[91,3] = PR[90,3] + 20.471;
   1:L PR[91] R[100]mm/sec CNT100;
   1:  PR[91,1] = PR[90,1] + 16.307;
   1:  PR[91,2] = PR[90,2] + 17.856;
   1:  PR[91,3] = PR[90,3] + 20.476;
   1:L PR[91] R[100]mm/sec CNT100;
   1:  PR[91,1] = PR[90,1] + 15.149;
   1:  PR[91,2] = PR[90,2] + 17.796;
   1:  PR[91,3] = PR[90,3] + 20.484;
   1:L PR[91] R[100]mm/sec CNT100;
   1:  PR[91,1] = PR[90,1] + 14.437;
   1:  PR[91,2] = PR[90,2] + 17.729;
   1:  PR[91,3] = PR[90,3] + 20.492;
   1:L PR[91] R[100]mm/sec CNT100;
   1:  PR[91,1] = PR[90,1] + 13.514;
   1:  PR[91,2] = PR[90,2] + 17.600;
   1:  PR[91,3] = PR[90,3] + 20.497;
   1:L PR[91] R[100]mm/sec CNT100;
   1:  PR[91,1] = PR[90,1] + 12.458;
   1:  PR[91,2] = PR[90,2] + 17.396;
   1:  PR[91,3] = PR[90,3] + 20.504;
   1:L PR[91] R[100]mm/sec CNT100;
   1:  PR[91,1] = PR[90,1] + 11.638;
   1:  PR[91,2] = PR[90,2] + 17.197;
   1:  PR[91,3] = PR[90,3] + 20.511;
   1:L PR[91] R[100]mm/sec CNT100;
   1:  PR[91,1] = PR[90,1] + 10.925;
   1:  PR[91,2] = PR[90,2] + 16.993;
   1:  PR[91,3] = PR[90,3] + 20.517;
   1:L PR[91] R[100]mm/sec CNT100;
   1:  PR[91,1] = PR[90,1] + 10.302;
   1:  PR[91,2] = PR[90,2] + 16.790;
   1:  PR[91,3] = PR[90,3] + 20.522;
   1:L PR[91] R[100]mm/sec CNT100;
   1:  PR[91,1] = PR[90,1] + 9.725;
   1:  PR[91,2] = PR[90,2] + 16.582;
   1:  PR[91,3] = PR[90,3] + 20.527;
   1:L PR[91] R[100]mm/sec CNT100;
   1:  PR[91,1] = PR[90,1] + 9.095;
   1:  PR[91,2] = PR[90,2] + 16.332;
   1:  PR[91,3] = PR[90,3] + 20.531;
   1:L PR[91] R[100]mm/sec CNT100;
   1:  PR[91,1] = PR[90,1] + 8.559;
   1:  PR[91,2] = PR[90,2] + 16.099;
   1:  PR[91,3] = PR[90,3] + 20.536;
   1:L PR[91] R[100]mm/sec CNT100;
   1:  PR[91,1] = PR[90,1] + 7.938;
   1:  PR[91,2] = PR[90,2] + 15.804;
   1:  PR[91,3] = PR[90,3] + 20.540;
   1:L PR[91] R[100]mm/sec CNT100;
   1:  PR[91,1] = PR[90,1] + 7.298;
   1:  PR[91,2] = PR[90,2] + 15.469;
   1:  PR[91,3] = PR[90,3] + 20.545;
   1:L PR[91] R[100]mm/sec CNT100;
   1:  PR[91,1] = PR[90,1] + 6.880;
   1:  PR[91,2] = PR[90,2] + 15.235;
   1:  PR[91,3] = PR[90,3] + 20.550;
   1:L PR[91] R[100]mm/sec CNT100;
   1:  PR[91,1] = PR[90,1] + 6.258;
   1:  PR[91,2] = PR[90,2] + 14.859;
   1:  PR[91,3] = PR[90,3] + 20.554;
   1:L PR[91] R[100]mm/sec CNT100;
   1:  PR[91,1] = PR[90,1] + 5.302;
   1:  PR[91,2] = PR[90,2] + 14.211;
   1:  PR[91,3] = PR[90,3] + 20.559;
   1:L PR[91] R[100]mm/sec CNT100;
   1:  PR[91,1] = PR[90,1] + 4.697;
   1:  PR[91,2] = PR[90,2] + 13.753;
   1:  PR[91,3] = PR[90,3] + 20.567;
   1:L PR[91] R[100]mm/sec CNT100;
   1:  PR[91,1] = PR[90,1] + 3.853;
   1:  PR[91,2] = PR[90,2] + 13.042;
   1:  PR[91,3] = PR[90,3] + 20.572;
   1:L PR[91] R[100]mm/sec CNT100;
   1:  PR[91,1] = PR[90,1] + 3.082;
   1:  PR[91,2] = PR[90,2] + 12.305;
   1:  PR[91,3] = PR[90,3] + 20.580;
   1:L PR[91] R[100]mm/sec CNT100;
   1:  PR[91,1] = PR[90,1] + 2.529;
   1:  PR[91,2] = PR[90,2] + 11.718;
   1:  PR[91,3] = PR[90,3] + 20.587;
   1:L PR[91] R[100]mm/sec CNT100;
   1:  PR[91,1] = PR[90,1] + 2.059;
   1:  PR[91,2] = PR[90,2] + 11.165;
   1:  PR[91,3] = PR[90,3] + 20.593;
   1:L PR[91] R[100]mm/sec CNT100;
   1:  PR[91,1] = PR[90,1] + 1.691;
   1:  PR[91,2] = PR[90,2] + 10.812;
   1:  PR[91,3] = PR[90,3] + 20.598;
   1:L PR[91] R[100]mm/sec CNT100;
   1:  PR[91,1] = PR[90,1] + 1.261;
   1:  PR[91,2] = PR[90,2] + 10.521;
   1:  PR[91,3] = PR[90,3] + 20.602;
   1:L PR[91] R[100]mm/sec CNT100;
   1:  PR[91,1] = PR[90,1] + 0.793;
   1:  PR[91,2] = PR[90,2] + 10.311;
   1:  PR[91,3] = PR[90,3] + 20.605;
   1:L PR[91] R[100]mm/sec CNT100;
   1:  PR[91,1] = PR[90,1] + 0.301;
   1:  PR[91,2] = PR[90,2] + 10.191;
   1:  PR[91,3] = PR[90,3] + 20.609;
   1:L PR[91] R[100]mm/sec CNT100;
   1:  PR[91,1] = PR[90,1] + -0.199;
   1:  PR[91,2] = PR[90,2] + 10.161;
   1:  PR[91,3] = PR[90,3] + 20.613;
   1:L PR[91] R[100]mm/sec CNT100;
   1:  PR[91,1] = PR[90,1] + -0.694;
   1:  PR[91,2] = PR[90,2] + 10.220;
   1:  PR[91,3] = PR[90,3] + 20.616;
   1:L PR[91] R[100]mm/sec CNT100;
   1:  PR[91,1] = PR[90,1] + -1.170;
   1:  PR[91,2] = PR[90,2] + 10.368;
   1:  PR[91,3] = PR[90,3] + 20.620;
   1:L PR[91] R[100]mm/sec CNT100;
   1:  PR[91,1] = PR[90,1] + -1.614;
   1:  PR[91,2] = PR[90,2] + 10.593;
   1:  PR[91,3] = PR[90,3] + 20.623;
   1:L PR[91] R[100]mm/sec CNT100;
   1:  PR[91,1] = PR[90,1] + -2.018;
   1:  PR[91,2] = PR[90,2] + 10.892;
   1:  PR[91,3] = PR[90,3] + 20.627;
   1:L PR[91] R[100]mm/sec CNT100;
   1:  PR[91,1] = PR[90,1] + -2.350;
   1:  PR[91,2] = PR[90,2] + 11.238;
   1:  PR[91,3] = PR[90,3] + 20.630;
   1:L PR[91] R[100]mm/sec CNT100;
   1:  PR[91,1] = PR[90,1] + -2.752;
   1:  PR[91,2] = PR[90,2] + 11.708;
   1:  PR[91,3] = PR[90,3] + 20.634;
   1:L PR[91] R[100]mm/sec CNT100;
   1:  PR[91,1] = PR[90,1] + -3.305;
   1:  PR[91,2] = PR[90,2] + 12.292;
   1:  PR[91,3] = PR[90,3] + 20.638;
   1:L PR[91] R[100]mm/sec CNT100;
   1:  PR[91,1] = PR[90,1] + -4.074;
   1:  PR[91,2] = PR[90,2] + 13.026;
   1:  PR[91,3] = PR[90,3] + 20.644;
   1:L PR[91] R[100]mm/sec CNT100;
   1:  PR[91,1] = PR[90,1] + -4.920;
   1:  PR[91,2] = PR[90,2] + 13.738;
   1:  PR[91,3] = PR[90,3] + 20.651;
   1:L PR[91] R[100]mm/sec CNT100;
   1:  PR[91,1] = PR[90,1] + -5.528;
   1:  PR[91,2] = PR[90,2] + 14.199;
   1:  PR[91,3] = PR[90,3] + 20.659;
   1:L PR[91] R[100]mm/sec CNT100;
   1:  PR[91,1] = PR[90,1] + -6.133;
   1:  PR[91,2] = PR[90,2] + 14.617;
   1:  PR[91,3] = PR[90,3] + 20.664;
   1:L PR[91] R[100]mm/sec CNT100;
   1:  PR[91,1] = PR[90,1] + -7.113;
   1:  PR[91,2] = PR[90,2] + 15.229;
   1:  PR[91,3] = PR[90,3] + 20.669;
   1:L PR[91] R[100]mm/sec CNT100;
   1:  PR[91,1] = PR[90,1] + -8.183;
   1:  PR[91,2] = PR[90,2] + 15.806;
   1:  PR[91,3] = PR[90,3] + 20.678;
   1:L PR[91] R[100]mm/sec CNT100;
   1:  PR[91,1] = PR[90,1] + -8.802;
   1:  PR[91,2] = PR[90,2] + 16.101;
   1:  PR[91,3] = PR[90,3] + 20.686;
   1:L PR[91] R[100]mm/sec CNT100;
   1:  PR[91,1] = PR[90,1] + -9.405;
   1:  PR[91,2] = PR[90,2] + 16.362;
   1:  PR[91,3] = PR[90,3] + 20.691;
   1:L PR[91] R[100]mm/sec CNT100;
   1:  PR[91,1] = PR[90,1] + -9.970;
   1:  PR[91,2] = PR[90,2] + 16.586;
   1:  PR[91,3] = PR[90,3] + 20.696;
   1:L PR[91] R[100]mm/sec CNT100;
   1:  PR[91,1] = PR[90,1] + -10.545;
   1:  PR[91,2] = PR[90,2] + 16.794;
   1:  PR[91,3] = PR[90,3] + 20.700;
   1:L PR[91] R[100]mm/sec CNT100;
   1:  PR[91,1] = PR[90,1] + -11.164;
   1:  PR[91,2] = PR[90,2] + 16.995;
   1:  PR[91,3] = PR[90,3] + 20.704;
   1:L PR[91] R[100]mm/sec CNT100;
   1:  PR[91,1] = PR[90,1] + -12.202;
   1:  PR[91,2] = PR[90,2] + 17.281;
   1:  PR[91,3] = PR[90,3] + 20.709;
   1:L PR[91] R[100]mm/sec CNT100;
   1:  PR[91,1] = PR[90,1] + -12.923;
   1:  PR[91,2] = PR[90,2] + 17.446;
   1:  PR[91,3] = PR[90,3] + 20.716;
   1:L PR[91] R[100]mm/sec CNT100;
   1:  PR[91,1] = PR[90,1] + -13.744;
   1:  PR[91,2] = PR[90,2] + 17.599;
   1:  PR[91,3] = PR[90,3] + 20.722;
   1:L PR[91] R[100]mm/sec CNT100;
   1:  PR[91,1] = PR[90,1] + -14.668;
   1:  PR[91,2] = PR[90,2] + 17.728;
   1:  PR[91,3] = PR[90,3] + 20.727;
   1:L PR[91] R[100]mm/sec CNT100;
   1:  PR[91,1] = PR[90,1] + -15.605;
   1:  PR[91,2] = PR[90,2] + 17.814;
   1:  PR[91,3] = PR[90,3] + 20.734;
   1:L PR[91] R[100]mm/sec CNT100;
   1:  PR[91,1] = PR[90,1] + -16.543;
   1:  PR[91,2] = PR[90,2] + 17.856;
   1:  PR[91,3] = PR[90,3] + 20.741;
   1:L PR[91] R[100]mm/sec CNT100;
   1:  PR[91,1] = PR[90,1] + -16.945;
   1:  PR[91,2] = PR[90,2] + 17.857;
   1:  PR[91,3] = PR[90,3] + 20.747;
   1:L PR[91] R[100]mm/sec CNT100;
   1:  PR[91,1] = PR[90,1] + -17.474;
   1:  PR[91,2] = PR[90,2] + 17.853;
   1:  PR[91,3] = PR[90,3] + 20.750;
   1:L PR[91] R[100]mm/sec CNT100;
   1:  PR[91,1] = PR[90,1] + -18.404;
   1:  PR[91,2] = PR[90,2] + 17.805;
   1:  PR[91,3] = PR[90,3] + 20.754;
   1:L PR[91] R[100]mm/sec CNT100;
   1:  PR[91,1] = PR[90,1] + -19.299;
   1:  PR[91,2] = PR[90,2] + 17.718;
   1:  PR[91,3] = PR[90,3] + 20.760;
   1:L PR[91] R[100]mm/sec CNT100;
   1:  PR[91,1] = PR[90,1] + -20.334;
   1:  PR[91,2] = PR[90,2] + 17.563;
   1:  PR[91,3] = PR[90,3] + 20.767;
   1:L PR[91] R[100]mm/sec CNT100;
   1:  PR[91,1] = PR[90,1] + -21.312;
   1:  PR[91,2] = PR[90,2] + 17.364;
   1:  PR[91,3] = PR[90,3] + 20.774;
   1:L PR[91] R[100]mm/sec CNT100;
   1:  PR[91,1] = PR[90,1] + -22.277;
   1:  PR[91,2] = PR[90,2] + 17.115;
   1:  PR[91,3] = PR[90,3] + 20.781;
   1:L PR[91] R[100]mm/sec CNT100;
   1:  PR[91,1] = PR[90,1] + -23.226;
   1:  PR[91,2] = PR[90,2] + 16.818;
   1:  PR[91,3] = PR[90,3] + 20.788;
   1:L PR[91] R[100]mm/sec CNT100;
   1:  PR[91,1] = PR[90,1] + -24.202;
   1:  PR[91,2] = PR[90,2] + 16.454;
   1:  PR[91,3] = PR[90,3] + 20.795;
   1:L PR[91] R[100]mm/sec CNT100;
   1:  PR[91,1] = PR[90,1] + -25.013;
   1:  PR[91,2] = PR[90,2] + 16.102;
   1:  PR[91,3] = PR[90,3] + 20.802;
   1:L PR[91] R[100]mm/sec CNT100;
   1:  PR[91,1] = PR[90,1] + -25.820;
   1:  PR[91,2] = PR[90,2] + 15.705;
   1:  PR[91,3] = PR[90,3] + 20.809;
   1:L PR[91] R[100]mm/sec CNT100;
   1:  PR[91,1] = PR[90,1] + -26.604;
   1:  PR[91,2] = PR[90,2] + 15.272;
   1:  PR[91,3] = PR[90,3] + 20.815;
   1:L PR[91] R[100]mm/sec CNT100;
   1:  PR[91,1] = PR[90,1] + -27.362;
   1:  PR[91,2] = PR[90,2] + 14.803;
   1:  PR[91,3] = PR[90,3] + 20.821;
   1:L PR[91] R[100]mm/sec CNT100;
   1:  PR[91,1] = PR[90,1] + -28.093;
   1:  PR[91,2] = PR[90,2] + 14.302;
   1:  PR[91,3] = PR[90,3] + 20.828;
   1:L PR[91] R[100]mm/sec CNT100;
   1:  PR[91,1] = PR[90,1] + -28.346;
   1:  PR[91,2] = PR[90,2] + 14.111;
   1:  PR[91,3] = PR[90,3] + 20.834;
   1:L PR[91] R[100]mm/sec CNT100;
   1:  PR[91,1] = PR[90,1] + -28.794;
   1:  PR[91,2] = PR[90,2] + 13.769;
   1:  PR[91,3] = PR[90,3] + 20.836;
   1:L PR[91] R[100]mm/sec CNT100;
   1:  PR[91,1] = PR[90,1] + -29.466;
   1:  PR[91,2] = PR[90,2] + 13.205;
   1:  PR[91,3] = PR[90,3] + 20.840;
   1:L PR[91] R[100]mm/sec CNT100;
   1:  PR[91,1] = PR[90,1] + -30.107;
   1:  PR[91,2] = PR[90,2] + 12.611;
   1:  PR[91,3] = PR[90,3] + 20.846;
   1:L PR[91] R[100]mm/sec CNT100;
   1:  PR[91,1] = PR[90,1] + -30.717;
   1:  PR[91,2] = PR[90,2] + 11.987;
   1:  PR[91,3] = PR[90,3] + 20.852;
   1:L PR[91] R[100]mm/sec CNT100;
   1:  PR[91,1] = PR[90,1] + -31.286;
   1:  PR[91,2] = PR[90,2] + 11.340;
   1:  PR[91,3] = PR[90,3] + 20.858;
   1:L PR[91] R[100]mm/sec CNT100;
   1:  PR[91,1] = PR[90,1] + -31.822;
   1:  PR[91,2] = PR[90,2] + 10.665;
